IF xResetRequest//清空报警
THEN
	eERRORID := MT_MCK_ERROR.No_ERROR;
END_IF
IF  xAutoMode OR xDeviceRunning THEN
	xAutomodeFlag:=TRUE;
ELSE
	xAutomodeFlag:=FALSE;
END_IF


IF eErrorID = MT_MCK_ERROR.NO_ERROR AND xEStop 
THEN
//获取序列号
	IF(stDeviceOpe.xReadSerialNum_HMI AND NOT xAutomodeFlag) OR (stDeviceOpe.xReadSerialNum_Auto AND xAutomodeFlag) THEN
		eCmd := MT_MCK_CMD.Cmd_SerialNum;
		xExecute := TRUE;
	END_IF
//获取重量
	IF (stDeviceOpe.xAcquireWeight_Steady_HMI AND NOT xAutomodeFlag) OR (stDeviceOpe.xAcquireWeight_Steady_Auto AND xAutomodeFlag) THEN
		eCmd := MT_MCK_CMD.Cmd_AcquireWeight_Steady;
		xExecute := TRUE;		
	END_IF
	IF (stDeviceOpe.xAcquireWeight_RealTime_HMI AND NOT xAutomodeFlag) OR (stDeviceOpe.xAcquireWeight_RealTime_Auto AND xAutomodeFlag) THEN
		eCmd := MT_MCK_CMD.Cmd_AcquireWeight_RealTime;
		xExecute := TRUE;		
	END_IF	
	IF (stDeviceOpe.xAcquireWeight_Continuous_HMI AND NOT xAutomodeFlag) OR (stDeviceOpe.xAcquireWeight_Continuous_Auto AND xAutomodeFlag) THEN
		eCmd := MT_MCK_CMD.Cmd_AcquireWeight_Continuous;
		xExecute := TRUE;		
	END_IF	
	IF (stDeviceOpe.xAcquireWeight_Stop_HMI AND NOT xAutomodeFlag) OR (stDeviceOpe.xAcquireWeight_Stop_Auto AND xAutomodeFlag) THEN
		eCmd := MT_MCK_CMD.Cmd_AcquireWeight_Stop;
		xExecute := TRUE;		
	END_IF
//重启
	IF (stDeviceOpe.xRestart_HMI AND NOT xAutomodeFlag) OR (stDeviceOpe.xRestart_Auto AND xAutomodeFlag) THEN
		eCmd := MT_MCK_CMD.Cmd_Restart;
		xExecute := TRUE;		
	END_IF	
//去皮重
	IF (stDeviceOpe.xShelling_HMI AND NOT xAutomodeFlag) OR (stDeviceOpe.xShelling_Auto AND xAutomodeFlag) THEN
		eCmd := MT_MCK_CMD.Cmd_Shelling;
		xExecute := TRUE;		
	END_IF	
	IF (stDeviceOpe.xShellingInstanly_HMI AND NOT xAutomodeFlag) OR (stDeviceOpe.xShellingInstanly_Auto AND xAutomodeFlag) THEN
		eCmd := MT_MCK_CMD.Cmd_ShellingInstanly;
		xExecute := TRUE;		
	END_IF
	IF (stDeviceOpe.xSetTare_HMI AND NOT xAutomodeFlag) OR (stDeviceOpe.xSetTare_Auto AND xAutomodeFlag) THEN
		rTareSet:=stpar.rTarePresetValue;//
		eCmd := MT_MCK_CMD.Cmd_SetTare;
		xExecute := TRUE;		
	END_IF
	IF (stDeviceOpe.xlearTare_HMI AND NOT xAutomodeFlag) OR (stDeviceOpe.xlearTare_Auto AND xAutomodeFlag) THEN
		eCmd := MT_MCK_CMD.Cmd_ClearTare;
		xExecute := TRUE;		
	END_IF	
//清零
	IF (stDeviceOpe.xClearZero_HMI AND NOT xAutomodeFlag) OR (stDeviceOpe.xClearZero_Auto AND xAutomodeFlag) THEN
		eCmd := MT_MCK_CMD.Cmd_ClearZero;
		xExecute := TRUE;		
	END_IF	
	IF (stDeviceOpe.xClearZeroInstanly_HMI AND NOT xAutomodeFlag) OR (stDeviceOpe.xClearZeroInstanly_Auto AND xAutomodeFlag) THEN
		eCmd := MT_MCK_CMD.Cmd_ClearZeroInstanly;
		xExecute := TRUE;		
	END_IF		
	
END_IF
END_METHOD

{attribute 'tc_no_symbol'}
METHOD PRIVATE FINAL  HandleErrorSTATE
VAR_INPUT
END_VAR
VAR_OUTPUT
	xAgain: BOOL;
END_VAR
IF xError AND  (xResetRequest OR NOT xExecute) THEN
    eState:=STATE.RESETING;
    xAgain:=1;
ELSE
    xBusy:=0;
    xError:=1;    
    xAgain:=0;(* !!! *)
END_IF
END_METHOD

{attribute 'tc_no_symbol'}
METHOD PRIVATE FINAL HandleExecutingSTATE
VAR_INPUT
END_VAR
VAR_OUTPUT
	xAgain: BOOL;
END_VAR
VAR
{attribute 'tc_no_symbol'}	
	xComplete: BOOL;
END_VAR

IF xAbort=0 THEN   
    CyclicAction(xComplete=> xComplete);
END_IF

IF eErrorID<>MT_MCK_ERROR.NO_ERROR THEN
    eState:=STATE.INERROR;
    xAgain:=1;
ELSIF xAbort THEN
    eState:=STATE.ABORTING;
    xAgain:=1;
ELSIF xComplete THEN
    eState:=STATE.DONE;
    xAgain:=1;
END_IF
END_METHOD

{attribute 'tc_no_symbol'}
METHOD PRIVATE FINAL HandleResettingSTATE
VAR_INPUT
END_VAR
VAR_OUTPUT
	xAgain: BOOL;
END_VAR
VAR
{attribute 'tc_no_symbol'}	
	xComplete: BOOL;
END_VAR
ResetAction(xComplete=> xComplete);

IF xComplete THEN
		xExecute:=0;//清除输入指令 
    xBusy:=0;
    _xDone:=0;
    xError:=0;

    eErrorID:=MT_MCK_ERROR.NO_ERROR;
    eState:=STATE.DORMANT;
    xFirstInvocation:=1;
    xAgain:=0;(* !!! *)
END_IF
END_METHOD

{attribute 'tc_no_symbol'}
METHOD PROTECTED ResetAction
VAR_INPUT
END_VAR
VAR_OUTPUT
	xComplete: BOOL;
END_VAR
(*
* Cleaning
* => free all allocated resources
* => reinitialize instance variables
*)
tOperationTimer(IN:=0);
_tDelay(IN:=FALSE);
_iNGCount  := 0;
_fbTcpIpClient(xEnable:=FALSE);
_diCmdState:=0;
eCmd := MT_MCK_CMD.Nodef;

//复位操作按钮
	stDeviceOpe.xAcquireWeight_Continuous_Auto	:=
	stDeviceOpe.xAcquireWeight_Continuous_HMI	:=
	stDeviceOpe.xAcquireWeight_RealTime_Auto	:=
	stDeviceOpe.xAcquireWeight_RealTime_HMI		:=
	stDeviceOpe.xAcquireWeight_Steady_Auto		:=
	stDeviceOpe.xAcquireWeight_Steady_HMI		:=
	stDeviceOpe.xAcquireWeight_Stop_Auto		:=
	stDeviceOpe.xAcquireWeight_Stop_HMI			:=
	stDeviceOpe.xClearZero_Auto					:=
	stDeviceOpe.xClearZero_HMI                  :=
	stDeviceOpe.xClearZeroInstanly_Auto         :=
	stDeviceOpe.xClearZeroInstanly_HMI          :=
	stDeviceOpe.xlearTare_Auto                  :=
	stDeviceOpe.xlearTare_HMI                   :=
	stDeviceOpe.xReadSerialNum_Auto             :=
	stDeviceOpe.xReadSerialNum_HMI              :=
	stDeviceOpe.xRestart_Auto					:=
	stDeviceOpe.xRestart_HMI                    :=
	stDeviceOpe.xSetTare_Auto                   :=
	stDeviceOpe.xSetTare_HMI                    :=
	stDeviceOpe.xShelling_Auto                  :=
	stDeviceOpe.xShelling_HMI                   :=
	stDeviceOpe.xShellingInstanly_Auto          :=
	stDeviceOpe.xShellingInstanly_HMI           :=FALSE;

xComplete:=1;
END_METHOD

END_FUNCTION_BLOCK

// ---- POUs/003_FB/53_RudongPump/08_PeristalticPumpFB/校准程序/FB_AutoCal.TcPOU
{attribute 'tc_no_symbol'}
FUNCTION_BLOCK FB_AutoCal//METTLER电子秤
VAR_INPUT
	xExecute		: BOOL;//指令执行
	xAbort			: BOOL;//指令中断
	xEstop			: BOOL;//急停
	xDeviceRunning	: BOOL;
	xResetRequest	: BOOL;//复位操作
	stDeviceOpe		: ST_AutoCalOpe;
	stparIn				: STAutoCal_ParIn;	 
	stSysPar			: ST_AutoCal_SysPar; 
	xAutoMode    	: BOOL;//0:mannal 1:auto
	xIniting    	: BOOL;//初始化过程中  

END_VAR
VAR_OUTPUT
	xDone			: BOOL;(*完成条件满足*)
	xBusy			: BOOL;(*动作正在执行*)
	xRunning	: BOOL;
	xError			: BOOL;(*错误条件满足*)
	eERRORID		: AutoCal_ERROR;
	xRdyCmd			: BOOL;//指令就绪
	xRdy			: BOOL;//初始化完成
	sHmiError	:STRING;
	stParOut		: STAutoCal_ParOut;
END_VAR

VAR
{attribute 'tc_no_symbol'}
	eState: STATE;//当前状态
{attribute 'tc_no_symbol'}
	xAborted: BOOL;(*指令被打断，一般是处于急停中*)
{attribute 'tc_no_symbol'}
	_CalStep	:INT;//校准流程
{attribute 'tc_no_symbol'}
	_CurrentPumpController	:INT:=1;//当前控制器
{attribute 'tc_no_symbol'}
	_CurrentPumpHead	:INT:=1;//当前泵头
{attribute 'tc_no_symbol'}
	_first :BOOL;
{attribute 'tc_no_symbol'}		
	_xModeChange:BOOL;
{attribute 'tc_no_symbol'}
	_fManual:F_TRIG;
{attribute 'tc_no_symbol'}
	_rManual:R_TRIG;
{attribute 'tc_no_symbol'}	
	i:INT;
{attribute 'tc_no_symbol'}		
	xFirstInvocation:BOOL;
{attribute 'tc_no_symbol'}	
	xAutomodeFlag:BOOL;	
{attribute 'tc_no_symbol'}		
	_diCmdState:INT;
{attribute 'tc_no_symbol'}
	eCmd:AutoCal_CMD;
{attribute 'tc_no_symbol'}
	tOperationTimer:TON;
{attribute 'tc_no_symbol'}
	tSteadyTimer:TON;	
{attribute 'tc_no_symbol'}	
	_xAutoOpe:BOOL;
{attribute 'tc_no_symbol'}	
	_xHMIOpe:BOOL;
{attribute 'tc_no_symbol'}	
	_xDone:BOOL;
{attribute 'tc_no_symbol'}	
	_InjectNum	:INT;//
{attribute 'tc_no_symbol'}
	k	:INT;//
{attribute 'tc_no_symbol'}
	xRuDongPumpError	:BOOL;	
{attribute 'tc_no_symbol'}
OperR_TRIG:ARRAY[1..5] OF R_TRIG;	
END_VAR

VAR_TEMP
{attribute 'tc_no_symbol'}
	xAgain: BOOL;

END_VAR

VAR

END_VAR


IF NOT _first 
THEN
	_first := TRUE;

ELSE
	xAgain:=0;	
//检测是否允许指令控制(初始状态，没有报警发生)	
	xRdyCmd := eState = STATE.DORMANT AND eERRORID = AutoCal_ERROR.No_ERROR;
	xDone:=_xDone AND xExecute;	
	//检测是否有模式变化
_fManual(CLK:=xAutoMode);
_rManual(CLK:=xAutoMode);
//

IF eState <> STATE.DORMANT//只有在运行的时候，才会检测是否有模式切换发生
THEN
	IF _fManual.Q OR _rManual.Q
	THEN
		_xModeChange := TRUE;
	END_IF
END_IF
	REPEAT
		CASE eState OF
			STATE.DORMANT:
				HandleDormantState(xAgain=> xAgain);
			STATE.EXECUTING:
				HandleExecutingState(xAgain=> xAgain);
			STATE.DONE:
				HandleDoneState(xAgain=> xAgain);
			STATE.INERROR:
				HandleErrorState(xAgain=> xAgain);
			STATE.ABORTING:
				HandleAbortingState(xAgain=> xAgain);
			STATE.ABORTED:
				HandleAbortedState(xAgain=> xAgain);
			STATE.RESETING:
				HandleResettingState(xAgain=> xAgain);
			END_CASE
	UNTIL (xAgain=0)
	END_REPEAT
END_IF


//报错内容输出
CASE eERRORID OF
	AutoCal_ERROR.FLT_AutoMode:
		sHmiError:='FLT_AutoMode';
	AutoCal_ERROR.FLT_CmdTimeOut:
		sHmiError:='FLT_CmdTimeOut';	
	AutoCal_ERROR.FLT_MT_MCK204C:
		sHmiError:='FLT_MT_MCK204C';	
	AutoCal_ERROR.FLT_PARA:
		sHmiError:='FLT_PARA';	
	AutoCal_ERROR.FLT_RudongPump:
		sHmiError:='FLT_RudongPump';	
	AutoCal_ERROR.No_ERROR:
		sHmiError:='No_ERROR';
END_CASE




_xAutoOpe:=stDeviceOpe.x96PumpHeadCal_Auto OR
					stDeviceOpe.xSpecificPumpHeadCal_Auto;
_xHMIOpe:=stDeviceOpe.x96PumpHeadCal_HMI OR
					stDeviceOpe.xContinuesInject_HMI OR
					stDeviceOpe.xInit_Hmi OR
					stDeviceOpe.xSpecificPumpHeadCal_HMI;

{attribute 'tc_no_symbol'}
METHOD PROTECTED AbortAction
VAR_INPUT
END_VAR
VAR_OUTPUT
	xComplete: BOOL;
	eErrorID: AutoCal_ERROR;
END_VAR
(*
* Cleaning
* => abort all running operation
* => if an NBS.ERROR codition is reached, set eErrorID to a Value rather then NBS.ERROR.NO_ERROR 
*)
xComplete:=1;
eErrorID:=AutoCal_ERROR.NO_ERROR;
END_METHOD

ACTION ACT_DensityConversion:
{attribute 'tc_no_symbol'}
//密度计算公式，ρ＝m/V 
IF stParIn.rDensity<>0 THEN
	stParOut.rVolume:=stParOut.rSteadyWeight/stParIn.rDensity;
ELSE
	stParOut.rVolume:=0;
END_IF
END_ACTION

METHOD PROTECTED Cmd_ContinuesInject : BOOL
VAR_INPUT
END_VAR
VAR_OUTPUT
	xComplete: BOOL;
END_VAR
// return the real actual fault number
IF eERRORID <> AutoCal_ERROR.No_ERROR
THEN
  RETURN;  
END_IF
stParOut.iCalStep:=_diCmdState;//流程步输出

CASE _diCmdState OF	
	
		
	0://判断是否到达校准位置
		_diCmdState:=_diCmdState+1;	
			
	1://判断是否结束
	IF _InjectNum<=stparIn.iContinuesInjectNum THEN
		_diCmdState:=_diCmdState+1;
	ELSE
		_diCmdState:=30;//结束加液
	END_IF				
	
	2://等待秤Ready
		IF stsyspar.fbMTMCK204C^.xRdyCmd AND stsyspar.fbRuDongPump[stparIn.iPumpController-1].xRdyCmd THEN
			_diCmdState:=_diCmdState+1;	
		END_IF
	
	3://秤体清零
		stsyspar.fbMTMCK204C^.stDeviceOpe.xShelling_Auto:=TRUE;
			_diCmdState:=_diCmdState+1;
	4://等待清零完成
		IF stsyspar.fbMTMCK204C^.xQDone THEN
			_diCmdState:=_diCmdState+1;
		END_IF

	5://等待稳定时间
		tSteadyTimer(IN:=stsyspar.fbMTMCK204C^.xRdyCmd,PT:=T#1S);
		IF tSteadyTimer.Q THEN
			tSteadyTimer(IN:=FALSE);
			_diCmdState:=_diCmdState+1;
		END_IF	
	
	6://蠕动泵加液
		stsyspar.fbRuDongPump[stparIn.iPumpController-1].stDeviceOpe.xPush_Auto[1]:=TRUE;
		IF stsyspar.fbRuDongPump[stparIn.iPumpController-1].xDone THEN
			stsyspar.fbRuDongPump[stparIn.iPumpController-1].xExecute:=FALSE;
			_diCmdState:=_diCmdState+1;
		END_IF

	7://等待稳定时间
		tSteadyTimer(IN:=stsyspar.fbRuDongPump[stparIn.iPumpController-1].xRdyCmd,PT:=TO_TIME((stparIn.tSteadyTime +stsyspar.fbRuDongPump[stparIn.iPumpController-1].stRunPara.rPushRuntime[1])*1000 ));
		IF tSteadyTimer.Q THEN
			tSteadyTimer(IN:=FALSE);
			_diCmdState:=_diCmdState+1;
		END_IF
	
	8://读取重量
		stsyspar.fbMTMCK204C^.stDeviceOpe.xAcquireWeight_Steady_Auto:=TRUE;
			_diCmdState:=_diCmdState+1;
	9://等待读取完成
					IF stsyspar.fbMTMCK204C^.xQDone THEN
								_diCmdState:=_diCmdState+1;
					END_IF
	10://等待稳定时间
		tSteadyTimer(IN:=stsyspar.fbMTMCK204C^.xRdyCmd,PT:=T#1S);
		IF tSteadyTimer.Q THEN
			tSteadyTimer(IN:=FALSE);
			_diCmdState:=_diCmdState+1;
		END_IF		
		
	11://传递重量值
		IF stsyspar.fbMTMCK204C^.stParOut.rCurrentWeight>0 THEN
			stParOut.rContinuesInjectWeight[_InjectNum]:=stsyspar.fbMTMCK204C^.stParOut.rCurrentWeight;
			IF stParOut.rContinuesInjectWeight[_InjectNum]=stsyspar.fbMTMCK204C^.stParOut.rCurrentWeight THEN
				_diCmdState:=_diCmdState+1;
			END_IF
		ELSE
			_diCmdState:=8;
		END_IF		
	
	12://累加
		_InjectNum:=_InjectNum+1;
		_diCmdState:=_diCmdState+1;
	
	13://复位状态
		tSteadyTimer(IN:=TRUE,PT:=T#1S);
		IF tSteadyTimer.Q THEN
			tSteadyTimer(IN:=FALSE);
			_diCmdState:=0;
		END_IF	
		
		
(**************************************************加液结束***************************************************)	
	30://校准完成
		xComplete:=TRUE;
		
	
	
	
	
END_CASE
END_METHOD

METHOD PROTECTED Cmd_Init : BOOL
VAR_INPUT
END_VAR
VAR_OUTPUT
	xComplete: BOOL;
END_VAR
// return the real actual fault number
IF eERRORID <> AutoCal_ERROR.No_ERROR
THEN
  RETURN;  
END_IF
stParOut.iCalStep:=_diCmdState;//流程步输出
CASE _diCmdState OF	
		
	0://
		_CurrentPumpController:=1;//从1#泵开始
		_diCmdState:=10;
(**************蠕动泵停止**************)			
	10://判断N#泵控制器参数
		_CurrentPumpController:=1;//从1#开始
		_diCmdState:=_diCmdState+1;
		
	11://判断是否结束
		IF	_CurrentPumpController>=gc_uiRudongPump THEN
			_diCmdState:=20;
		ELSE
		 stSysPar.fbRuDongPump[_CurrentPumpController-1].xExecute:=FALSE;
			IF stSysPar.fbRuDongPump[_CurrentPumpController-1].xRdyCmd THEN
				_diCmdState:=_diCmdState+1;
			END_IF
		END_IF
		
	12://停止N#泵控制器	
		stSysPar.fbRuDongPump[_CurrentPumpController-1].stDeviceOpe.xStop_Auto:=TRUE;
				_diCmdState:=_diCmdState+1;
	13://等待停止	
					IF stSysPar.fbRuDongPump[_CurrentPumpController-1].xDone THEN
					 stSysPar.fbRuDongPump[_CurrentPumpController-1].stDeviceOpe.xStop_Auto:=FALSE;
						stSysPar.fbRuDongPump[_CurrentPumpController-1].xExecute:=FALSE;
						_diCmdState:=_diCmdState+1;
					END_IF	
	14://累加1
		_CurrentPumpController:=_CurrentPumpController+1;
		_diCmdState:=_diCmdState+1;
		
	15://回去循环执行
		_diCmdState:=11;

(**************************************************秤清零***************************************************)	
	20://判断秤体状态
		IF stSysPar.fbMTMCK204C^.xRdyCmd THEN
			_diCmdState:=22;
		ELSE
			IF stSysPar.fbMTMCK204C^.stParOut.xContinuesRead THEN
				_diCmdState:=_diCmdState+1;
			END_IF
		END_IF
	
	21://停止连续读取
			stSysPar.fbMTMCK204C^.stDeviceOpe.xAcquireWeight_Stop_Auto:=TRUE;
			IF stSysPar.fbMTMCK204C^.xRdyCmd THEN
				_diCmdState:=_diCmdState+1;
			END_IF			

	22://秤清零
			stSysPar.fbMTMCK204C^.stDeviceOpe.xClearZeroInstanly_Auto:=TRUE;
			_diCmdState:=_diCmdState+1;
	23://称清零完成
			IF stSysPar.fbMTMCK204C^.xQDone THEN
				_diCmdState:=30;
			END_IF			
	

(*************************************************初始化结束***************************************************)
	30://校准完成
		xComplete:=TRUE;
		

	
END_CASE
END_METHOD

METHOD PROTECTED Cmd_SpecificPumpHeadCal : BOOL
VAR_INPUT
END_VAR
VAR_OUTPUT
	xComplete: BOOL;
END_VAR
// return the real actual fault number
IF eERRORID <> AutoCal_ERROR.No_ERROR
THEN
  RETURN;  
END_IF
stParOut.iCalStep:=_diCmdState;//流程步输出

CASE _diCmdState OF	
	
		
	0://判断是否到达校准位置
		_diCmdState:=_diCmdState+1;	
		
	1://等待校准就绪
		stsyspar.fbRuDongPump[stparIn.iPumpController-1].xExecute:=FALSE;
		IF stsyspar.fbMTMCK204C^.xQRdyCmd AND stsyspar.fbRuDongPump[stparIn.iPumpController-1].xRdyCmd THEN
			_diCmdState:=_diCmdState+1;	

		END_IF		
		
(**************************************************校准***************************************************)		
	2://秤体清零	
		stSysPar.fbMTMCK204C^.stDeviceOpe.xClearZero_Auto:=TRUE;
			_diCmdState:=_diCmdState+1;	
	3://清零完成
		IF stSysPar.fbMTMCK204C^.xQDone THEN
			_diCmdState:=_diCmdState+1;	
		END_IF
		
	4://等待稳定时间
		tSteadyTimer(IN:=TRUE,PT:=T#1S);
		IF tSteadyTimer.Q THEN
			tSteadyTimer(IN:=FALSE);
			_diCmdState:=_diCmdState+1;
		END_IF		
		
	5://校准启动
		stSysPar.fbRuDongPump[_CurrentPumpController-1].stDeviceOpe.xPumpCal_Auto:=TRUE;
		IF stSysPar.fbRuDongPump[_CurrentPumpController-1].xDone THEN
		 	stSysPar.fbRuDongPump[_CurrentPumpController-1].xExecute:=FALSE;
			_diCmdState:=_diCmdState+1;
		END_IF
		
	6://等待稳定时间
		tSteadyTimer(IN:=TRUE,PT:=TO_TIME((stparIn.tSteadyTime+1)*1000));
		IF tSteadyTimer.Q THEN
			_diCmdState:=_diCmdState+1;
		END_IF

	7://获取称重结果
			stSysPar.fbMTMCK204C^.stDeviceOpe.xAcquireWeight_Steady_Auto:=TRUE;
				_diCmdState:=_diCmdState+1;
	8://等待完成
			IF stSysPar.fbMTMCK204C^.xQDone THEN
				_diCmdState:=_diCmdState+1;	
			END_IF	
	
	9://等待稳定时间
		tSteadyTimer(IN:=TRUE,PT:=T#1S);
		IF tSteadyTimer.Q THEN
			tSteadyTimer(IN:=FALSE);
			_diCmdState:=_diCmdState+1;
		END_IF			

	10://获取称重结果
		IF stSysPar.fbMTMCK204C^.stParOut.rCurrentWeight>0 THEN
			stParOut.rSteadyWeight:=stSysPar.fbMTMCK204C^.stParOut.rCurrentWeight;
			IF stParOut.rSteadyWeight=stSysPar.fbMTMCK204C^.stParOut.rCurrentWeight THEN
				_diCmdState:=_diCmdState+1;
			END_IF
		ELSE
			_diCmdState:=7;//未获取到重量重新读
		END_IF
		
	11://给校准参数赋值
		stSysPar.fbRuDongPump^.stRunPara.rModuleRealFluVolume:=stParOut.rVolume;
		stSysPar.fbRuDongPump^.stDeviceOpe.xCalParWrite_Auto:=TRUE;
		IF stSysPar.fbRuDongPump^.xDone THEN
			_diCmdState:=30;
		END_IF
	

(**************************************************校准结束***************************************************)	
	30://校准完成
		xComplete:=TRUE;
		
	
	
	
	
END_CASE
END_METHOD

{attribute 'tc_no_symbol'}
METHOD PROTECTED CyclicAction
VAR_INPUT
END_VAR
VAR_OUTPUT
	xComplete: BOOL;
END_VAR
VAR	
END_VAR
IF xAbort=0 THEN
	IF xFirstInvocation THEN//执行初始化
	(*
	* Staring
	* for then first (!) invocaion,
	* sample then input variables
	*)
		xFirstInvocation:=0;
	END_IF    
	REPEAT 	
//判断是否有参数错误		
		IF stSysPar.fbMTMCK204C=0 OR
				stSysPar.fbRuDongPump=0 OR
				stSysPar.iRuDongPumpHeadNum>32
		THEN
			eERRORID:=AutoCal_ERROR.FLT_PARA;//参数配置错误
		ELSE
			xRuDongPumpError:=FALSE;
			FOR k:=1 TO gc_uiRudongPump DO
				IF stSysPar.fbRuDongPump[k].xError THEN
					xRuDongPumpError:=TRUE;
					EXIT;
				END_IF
			END_FOR			

			//IF stSysPar.fbMTMCK204C^.xError THEN
			//	eERRORID:=AutoCal_ERROR.FLT_MT_MCK204C;//秤出错
			//ELSE
			//	IF xRuDongPumpError THEN
			//		eERRORID:=AutoCal_ERROR.FLT_RudongPump;//蠕动泵出错
			//	END_IF						
			//END_IF
		END_IF

			//如果不在自动模式则报错
			IF _xAutoOpe OR _xHMIOpe THEN
					xRunning:=TRUE;
			END_IF

			CASE eCmd OF//判断指令类型
				AutoCal_CMD.Cmd_SpecificPumpHeadCal://单个泵头校准
					Cmd_SpecificPumpHeadCal(xComplete=> xComplete);	
				AutoCal_CMD.Cmd_Init://初始化
					Cmd_Init(xComplete=> xComplete);	
				AutoCal_CMD.Cmd_ContinuesInject://连续加液测试
					Cmd_ContinuesInject(xComplete=> xComplete);
					;				
				
			ELSE
				;	
			END_CASE
	   
		UNTIL (TRUE)//处于一直刷新阶段
	END_REPEAT
END_IF

IF NOT xExecute OR xComplete OR eErrorID<>AutoCal_ERROR.No_ERROR THEN    
    (*
    * Cleaning
    * => free as much allocated resources as possible
    *)    
    tOperationTimer(IN:=0);
END_IF
END_METHOD

{attribute 'tc_no_symbol'}
METHOD PRIVATE FINAL HandleAbortedSTATE
VAR_INPUT
END_VAR
VAR_OUTPUT
	xAgain: BOOL;
END_VAR
VAR
	xComplete: BOOL;
END_VAR
IF xAborted AND xResetRequest THEN
    eState:=STATE.RESETING;
    xAgain:=1;
ELSE
    xBusy:=0;
    xAborted:=1;
    //xResetRequest:=(xExecute=0);
    xAgain:=0;(* !!! *)
END_IF
END_METHOD

{attribute 'tc_no_symbol'}
METHOD PRIVATE FINAL HandleAbortingSTATE
VAR_INPUT
END_VAR
VAR_OUTPUT
	xAgain: BOOL;
END_VAR
VAR
{attribute 'tc_no_symbol'}	
	xComplete: BOOL;
END_VAR
AbortAction(xComplete=> xComplete, eErrorID=> eErrorID);

IF eErrorID<>AutoCal_ERROR.NO_ERROR THEN
    eState:=STATE.INERROR;
    xAgain:=1;
ELSIF xComplete THEN
    eState:=STATE.ABORTED;
    xAgain:=1;
END_IF
END_METHOD

{attribute 'tc_no_symbol'}
METHOD PRIVATE FINAL HandleDoneSTATE
VAR_INPUT
END_VAR
VAR_OUTPUT
	xAgain: BOOL;
END_VAR
//在运行过程中要是切换模式，再运行完成之后，检测到模式的切换，就需要回到初始位置，进行下一次执行准备
IF _xDone AND ((xExecute=0) OR ( _xModeChange AND NOT _xAutoOpe)  OR ( NOT xAutoMode AND NOT xDeviceRunning AND ( NOT _xAutoOpe OR _xHMIOpe))) THEN
	eState:=STATE.RESETING;
	xAgain:=1;
ELSE
	xBusy:=0;
	_xDone:=1;
	//xResetRequest:=(xExecute=0);
	xAgain:=0;(* !!! *)
END_IF
END_METHOD

{attribute 'tc_no_symbol'}
METHOD PRIVATE FINAL HandleDormantSTATE
VAR_INPUT
END_VAR
VAR_OUTPUT
	xAgain: BOOL;
END_VAR
IF xExecute THEN
    xBusy:=1;
    eState:=STATE.EXECUTING;
    xAgain:=1;
END_IF

IF xResetRequest//清空报警
THEN
	eERRORID := AutoCal_ERROR.No_ERROR;
END_IF
IF  xAutoMode OR xDeviceRunning THEN
	xAutomodeFlag:=TRUE;
ELSE
	xAutomodeFlag:=FALSE;
END_IF
(********************************等待手动操作******************************)
OperR_TRIG[1](CLK:=  (stDeviceOpe.xSpecificPumpHeadCal_HMI OR stDeviceOpe.xSpecificPumpHeadCal_Auto) , Q=> );
OperR_TRIG[2](CLK:=  (stDeviceOpe.xInit_Hmi  OR stDeviceOpe.xInit_Auto)  , Q=> );

IF eErrorID = AutoCal_ERROR.NO_ERROR AND xEStop
THEN
	
//校准指定泵头
	IF OperR_TRIG[1].Q THEN//
		_CurrentPumpController:=stparIn.iPumpController;
		_CurrentPumpHead:=stparIn.iPumpHead;
		eCmd := AutoCal_CMD.Cmd_SpecificPumpHeadCal;
		xExecute := TRUE;
	END_IF
//初始化校准程序
	IF OperR_TRIG[2].Q THEN//
		eCmd := AutoCal_CMD.Cmd_Init;
		xExecute := TRUE;
	END_IF	
	
	
	
	stDeviceOpe.xSpecificPumpHeadCal_HMI := stDeviceOpe.xSpecificPumpHeadCal_Auto:=FALSE;
	stDeviceOpe.xInit_Hmi  := stDeviceOpe.xInit_Auto:=FALSE;
	
//连续加液测试
	IF stDeviceOpe.xContinuesInject_HMI THEN//
		FOR i:=1 TO 30 DO
			stParOut.rContinuesInjectWeight[i]:=0;
		END_FOR
		_InjectNum:=1;
		eCmd := AutoCal_CMD.Cmd_ContinuesInject;
		xExecute := TRUE;
	END_IF	
	
END_IF
END_METHOD

{attribute 'tc_no_symbol'}
METHOD PRIVATE FINAL  HandleErrorSTATE
VAR_INPUT
END_VAR
VAR_OUTPUT
	xAgain: BOOL;
END_VAR
IF xError AND  (xResetRequest OR NOT xExecute) THEN
    eState:=STATE.RESETING;
    xAgain:=1;
ELSE
    xBusy:=0;
    xError:=1;    
    xAgain:=0;(* !!! *)
END_IF
END_METHOD

{attribute 'tc_no_symbol'}
METHOD PRIVATE FINAL HandleExecutingSTATE
VAR_INPUT
END_VAR
VAR_OUTPUT
	xAgain: BOOL;
END_VAR
VAR
{attribute 'tc_no_symbol'}	
	xComplete: BOOL;
END_VAR

IF xAbort=0 THEN   
    CyclicAction(xComplete=> xComplete);
END_IF

IF eErrorID<>AutoCal_ERROR.NO_ERROR THEN
    eState:=STATE.INERROR;
    xAgain:=1;
ELSIF xAbort THEN
    eState:=STATE.ABORTING;
    xAgain:=1;
ELSIF xComplete THEN
    eState:=STATE.DONE;
    xAgain:=1;
END_IF
END_METHOD

{attribute 'tc_no_symbol'}
METHOD PRIVATE FINAL HandleResettingSTATE
VAR_INPUT
END_VAR
VAR_OUTPUT
	xAgain: BOOL;
END_VAR
VAR
{attribute 'tc_no_symbol'}	
	xComplete: BOOL;
END_VAR
ResetAction(xComplete=> xComplete);

IF xComplete THEN
		xExecute:=0;//清除输入指令 
    xBusy:=0;
    xDone:=0;
    xError:=0;

    eErrorID:=AutoCal_ERROR.NO_ERROR;
    eState:=STATE.DORMANT;
    xFirstInvocation:=1;
    xAgain:=0;(* !!! *)
END_IF
END_METHOD

{attribute 'tc_no_symbol'}
METHOD PROTECTED ResetAction
VAR_INPUT
END_VAR
VAR_OUTPUT
	xComplete: BOOL;
END_VAR
(*
* Cleaning
* => free all allocated resources
* => reinitialize instance variables
*)
tOperationTimer(IN:=0);
_diCmdState:=0;
_CurrentPumpController:=1;
stDeviceOpe.x96PumpHeadCal_Auto:=
stDeviceOpe.x96PumpHeadCal_HMI:=
stDeviceOpe.xInit_Auto:=
stDeviceOpe.xInit_Hmi:=
stDeviceOpe.xSpecificPumpHeadCal_Auto:=
stDeviceOpe.xContinuesInject_HMI:=
stDeviceOpe.xSpecificPumpHeadCal_HMI:=FALSE;
xRunning:=FALSE; 
xComplete:=1;	

stsyspar.fbRuDongPump[stparIn.iPumpController-1].xExecute:=FALSE;
//stsyspar.fbRuDongPump[stparIn.iPumpController-1].stDeviceOpe.xPush_Auto[1]:=TRUE;
stsyspar.fbRuDongPump[stparIn.iPumpController-1].stDeviceOpe.xStop_Auto:=TRUE;
END_METHOD

END_FUNCTION_BLOCK

// ---- POUs/003_FB/0015_Functions/FC_BubbleSort_Max.TcPOU
FUNCTION FC_BubbleSort_Max : REAL
(*
********************************************************************************
* Name: FB_BubbleSort_Max
*
* Author:  Automanh
* Version: 1.0.0
*
* Description:
*     将数组元素从小到大排列
*
* Remarks:
*
* Revisions:
*   1.0 -AutomanH Rebuild
*         
*  
*********************************************************************************)
VAR_INPUT
 i_i_Counter:INT;
 i_arrReal:ARRAY[1..3] OF REAL;
END_VAR
VAR
 i,j:INT;
 rRealTemp:REAL;
END_VAR


FOR i:=1 TO (i_i_Counter-1) BY 1 DO//控制比较轮次，一共 n-1 趟
 		FOR  j:=1 TO i_i_Counter-i BY 1 DO//控制两个挨着的元素进行比较
		 			IF i_arrReal[j]>i_arrReal[j+1] THEN
					 			rRealTemp:=i_arrReal[j];
								i_arrReal[j]:=i_arrReal[j+1];
								i_arrReal[j+1]:=rRealTemp;
					END_IF
		END_FOR
					
END_FOR
FC_BubbleSort_Max:=i_arrReal[i_i_Counter];

END_FUNCTION

// ---- POUs/003_FB/0015_Functions/FC_BubbleSort_Min.TcPOU
FUNCTION FC_BubbleSort_Min : REAL
(*
********************************************************************************
* Name: FB_BubbleSort_Min
*
* Author:  Automanh
* Version: 1.0.0
*
* Description:
*     将数组元素从大到小排列
*
* Remarks:
*
* Revisions:
*   1.0 -AutomanH Rebuild
*         
*  
*********************************************************************************)
VAR_INPUT
 i_i_Counter:INT;
 i_arrReal:ARRAY[1..3] OF REAL;
END_VAR
VAR
 i,j:INT;
 rRealTemp:REAL;
END_VAR

FOR i:=1 TO (i_i_Counter-1) BY 1 DO//控制比较轮次，一共 n-1 趟
 		FOR  j:=1 TO i_i_Counter-i BY 1 DO//控制两个挨着的元素进行比较
		 			IF i_arrReal[j]<i_arrReal[j+1] THEN
					 			rRealTemp:=i_arrReal[j];
								i_arrReal[j]:=i_arrReal[j+1];
								i_arrReal[j+1]:=rRealTemp;
					END_IF
		END_FOR
					
END_FOR
FC_BubbleSort_Min:=i_arrReal[i_i_Counter];

END_FUNCTION

// ---- POUs/001_Station/S03_LidChecking.TcPOU
PROGRAM S03_LidChecking
VAR
	//工站
	station					: REFERENCE TO FB_Station:=fbstation[3];
	//气缸
	fbHOZAdjustCyl_1	:REFERENCE TO FB_Cylinder:=fbCylinder[12];	//	上层水平调整气缸1（小）
	fbHOZAdjustCyl_2	:REFERENCE TO FB_Cylinder:=fbCylinder[13];	//	上层水平调整气缸2（小）
	fbHOZAdjustCyl_3	:REFERENCE TO FB_Cylinder:=fbCylinder[14];	//	下层水平调整气缸1（小）
	fbHOZAdjustCyl_4	:REFERENCE TO FB_Cylinder:=fbCylinder[15];	//	下层水平调整气缸2（小）
	fbHOZAdjustCyl_5	:REFERENCE TO FB_Cylinder:=fbCylinder[16];	//	上层水平调整气缸1（大）
	fbHOZAdjustCyl_6	:REFERENCE TO FB_Cylinder:=fbCylinder[17];	//	上层水平调整气缸2（大）
	fbHOZAdjustCyl_7	:REFERENCE TO FB_Cylinder:=fbCylinder[18];	//	下层水平调整气缸1（大）
	fbHOZAdjustCyl_8	:REFERENCE TO FB_Cylinder:=fbCylinder[19];	//	下层水平调整气缸2（大）
	//伺服
	fbXAxisMove	 :REFERENCE TO FB_Axis:=fbAxis[6];	//	相机检测工位X轴伺服
	fbYAxisMove	 :REFERENCE TO FB_Axis:=fbAxis[7];	//	相机检测工位Y轴伺服
	fbZAxisMove	 :REFERENCE TO FB_Axis:=fbAxis[8];	//	相机检测工位Z轴伺服
	//相机

	
		//延时
		arTonDelay :ARRAY[1..20] OF TON;
	//返回值
		UdiReturnValue :ARRAY[1..20] OF UDINT;
	//本地过程数据
	arProcessDataStation : ARRAY [1..5] OF DUT_MainlineFixture;
	
	i,j,k: INT;
	//循环使用
	i_b_REPEAT:BOOL;
	i_i_Counter:INT;
	//相机拍照结果步骤
	bResultStep:BYTE;
	// 循环计数
	bCounter: BYTE;
	// 临时变量
	_FirstCycle:ARRAY[1..10] OF BOOL;
	them: INT;
	// X轴伺服循环次数
	bXCounter: BYTE;
	// Y轴伺服循环次数
	bYCounter: BYTE;
	// 结束时循环次数
	bEndCounter: INT;
	//相机检测工位检测结果
	arCameraResult:ARRAY[1..5,1..4,1..12] OF INT;
	//过程记录
	tsModuleProcess:ARRAY[1..gc_ModuleProNo] OF DUT_Process;
	xClearModuleProcessDone:BOOL;
	bClearProcessStep	:BYTE;
	// 测试使用，待删
	xtest: BOOL;
	// //待删
	xnext: BOOL;
END_VAR

A_Input();
Alarm();
Delay();
FlowAuto();
FlowInit();
General();
ILC();
TipAuto();
TipManual();
Z_Output();

ACTION A_Input:
//气缸
//S03上层水平调整气缸1(小)
fbHOZAdjustCyl_1.xWP_Sensor	:=	IxS03HOZAdjustCyl_1WP	;
fbHOZAdjustCyl_1.xHP_Sensor	:=	IxS03HOZAdjustCyl_1HP 	;
//	上层水平调整气缸2（小）
fbHOZAdjustCyl_2.xWP_Sensor	:=	IxS03HOZAdjustCyl_2WP ;
fbHOZAdjustCyl_2.xHP_Sensor	:=	IxS03HOZAdjustCyl_2HP 	;

//S03下层水平调整气缸1(小)
fbHOZAdjustCyl_3.xWP_Sensor	:=	IxS03HOZAdjustCyl_5WP	;  
fbHOZAdjustCyl_3.xHP_Sensor	:=	IxS03HOZAdjustCyl_5HP ;
//下层水平调整气缸2（小）
fbHOZAdjustCyl_4.xWP_Sensor	:=	  IxS03HOZAdjustCyl_6WP;  
fbHOZAdjustCyl_4.xHP_Sensor	:=	  IxS03HOZAdjustCyl_6HP;
  
//S03上层水平调整气缸1(大）
fbHOZAdjustCyl_5.xWP_Sensor	:=IxS03HOZAdjustCyl_3WP ;										
fbHOZAdjustCyl_5.xHP_Sensor	:=IxS03HOZAdjustCyl_3HP	; 
//	上层水平调整气缸2（大）
fbHOZAdjustCyl_6.xWP_Sensor	:=IxS03HOZAdjustCyl_4WP ;										
fbHOZAdjustCyl_6.xHP_Sensor	:=IxS03HOZAdjustCyl_4HP	; 

//S03下层水平调整气缸1(大） 									 
fbHOZAdjustCyl_7.xWP_Sensor	:=	IxS03HOZAdjustCyl_7WP	;  
fbHOZAdjustCyl_7.xHP_Sensor	:=	IxS03HOZAdjustCyl_7HP	;  
//	下层水平调整气缸2（大）
fbHOZAdjustCyl_8.xWP_Sensor	:=		IxS03HOZAdjustCyl_8WP;  
fbHOZAdjustCyl_8.xHP_Sensor	:=		IxS03HOZAdjustCyl_8HP;
END_ACTION

ACTION Alarm:
station.adwAlarm[1].00	:=	station.xInitTimeout	;//	S03 初始化超时
station.adwAlarm[1].01	:=	fbHOZAdjustCyl_1.xHP_Off 	;//	S03上层水平调整气缸1(小)原点未到位
station.adwAlarm[1].02	:=	fbHOZAdjustCyl_1.xWP_Off 	;//	S03上层水平调整气缸1(小)动点未到位
station.adwAlarm[1].03	:=	fbHOZAdjustCyl_3.xHP_Off	;//	S03下层水平调整气缸1(小)原点未到位
station.adwAlarm[1].04	:=	fbHOZAdjustCyl_3.xWP_Off	;//	S03下层水平调整气缸1(小)动点未到位
station.adwAlarm[1].05	:=	fbHOZAdjustCyl_5.xHP_Off	;//	S03上层水平调整气缸1(大)原点未到位
station.adwAlarm[1].06	:=	fbHOZAdjustCyl_5.xWP_Off	;//	S03上层水平调整气缸1(大)动点未到位
station.adwAlarm[1].07	:=	fbHOZAdjustCyl_7.xHP_Off	;//	S03下层水平调整气缸1(大)原点未到位
station.adwAlarm[1].08	:=	fbHOZAdjustCyl_7.xWP_Off	;//	S03下层水平调整气缸1(大)动点未到位
station.adwAlarm[1].09	:=	fbXAxisMove.xError	;//	S03液位检测X轴伺服报错
station.adwAlarm[1].10	:=	fbXAxisMove.xNotPowerOn	;//	S03液位检测X轴伺服未使能
station.adwAlarm[1].11	:=	fbXAxisMove.xMoveTimeout	;//	S03液位检测X轴伺服移动超时
station.adwAlarm[1].12	:=	fbYAxisMove.xError	;//	S03液位检测Y轴伺服报错
station.adwAlarm[1].13	:=	fbYAxisMove.xNotPowerOn	;//	S03液位检测Y轴伺服未使能
station.adwAlarm[1].14	:=	fbYAxisMove.xMoveTimeout	;//	S03液位检测Y轴伺服移动超时
station.adwAlarm[1].15	:=	fbZAxisMove.xError	;//	S03液位检测Z轴伺服报错
station.adwAlarm[1].16	:=	fbZAxisMove.xNotPowerOn	;//	S03液位检测Z轴伺服未使能
station.adwAlarm[1].17	:=	fbZAxisMove.xMoveTimeout	;//	S03液位检测Z轴伺服移动超时
//station.adwAlarm[1].18	:=	true;//	S03液位检测工位-相机检测超时报警,请检查
END_ACTION

ACTION Delay:
arTonDelay[01](IN:= , PT:=T#0.1S , Q=> , ET=> );
arTonDelay[02](IN:=  , PT:=T#1S , Q=> , ET=> );
arTonDelay[03](IN:=   , PT:=T#1S , Q=> , ET=> );
arTonDelay[04](IN:= , PT:=T#0.1S , Q=> , ET=> );
arTonDelay[05](IN:= , PT:=T#0.1S , Q=> , ET=> );
arTonDelay[06](IN:= , PT:=T#0.1S , Q=> , ET=> );
(*arTonDelay[07](IN:= , PT:=T#200MS , Q=> , ET=> );*)//已使用
arTonDelay[08](IN:=NOT fbXAxisMove.xbusy , PT:=T#0.1S , Q=> , ET=> );//TipAuto使用
arTonDelay[09](IN:= NOT fbYAxisMove.xbusy, PT:=T#0.1S , Q=> , ET=> );//TipAuto使用
arTonDelay[10](IN:=NOT fbZAxisMove.xbusy , PT:=T#0.1S , Q=> , ET=> );//TipAuto使用
END_ACTION

ACTION FlowAuto:

//-----------------------------------------初始化是否完成判断----------------------------------------------
IF NOT station.xInitDone 
THEN
 	station.iStepAuto:=0;
 	station.xDone:=FALSE;
	station.xRunningOffProhibit := FALSE ;//运行中信号Off禁止
ELSIF station.xRunning // OR (tsModuleProcess[bXCounter+1].xProcessStarted AND NOT tsModuleProcess[bXCounter+1].xProcessCompleted )//相机检测流程
THEN
//-----------------------------------------动作步骤--------------------------------------------------------
CASE station.iStepAuto OF	  
	0: //----Home Step，等待启动----
		IF station.xDisabled 
			AND station.xCanRun 
			AND NOT fbMachine[1].xStopped 
			AND NOT station.xSingleRunning 
		THEN
			station.xDone:=TRUE;
		END_IF
		
		IF  station.xSingleRunning 
			OR station.xCanRun 
			AND NOT station.xDone 
			AND NOT station.xDisabled 
			AND NOT fbMachine[1].xStopped
		THEN
			station.xCycleEnable:=TRUE;
			station.xDone:= FALSE;  
			station.iStepAuto:= 5;
		END_IF		
	 5://复位数据
			FOR i:=1 TO gc_ModuleProNo BY 1 DO
				 MEMSET(ADR(tsModuleProcess[i]),0,SIZEOF(tsModuleProcess[i]));
			END_FOR
			station.iStepAuto:= 10;
	 10: //判断产品是否到该工位
		IF  station.xSingleRunning THEN
			station.iStepAuto:= 11;
		ELSE
		 			IF    station.xEmptyDone THEN
										station.iStepAuto:= 999;		
					//清料程序
					ELSIF   arMainlineFixtureData[arCurFixtureNumStation[5]].stProduct.xEmptying AND    
				    	arMainlineFixtureData[arCurFixtureNumStation[6]].stProduct.xEmptying  AND 
							arMainlineFixtureData[arCurFixtureNumStation[7]].xMaterialOnOff AND 
							arMainlineFixtureData[arCurFixtureNumStation[8]].xMaterialOnOff AND
							arMainlineFixtureData[arCurFixtureNumStation[9]].xMaterialOnOff  THEN
										 bEndCounter:=1;
										 bCounter:=0;
								 		 station.iStepAuto:= 11;
					ELSIF   arMainlineFixtureData[arCurFixtureNumStation[5]].stProduct.xEmptying AND    
									arMainlineFixtureData[arCurFixtureNumStation[6]].stProduct.xEmptying  AND 
									arMainlineFixtureData[arCurFixtureNumStation[7]].stProduct.xEmptying AND 
									arMainlineFixtureData[arCurFixtureNumStation[8]].stProduct.xEmptying AND
									arMainlineFixtureData[arCurFixtureNumStation[9]].xMaterialOnOff  THEN
												 bEndCounter:=2;
												 bCounter:=0;
												 station.iStepAuto:= 11;							 
					ELSIF   arMainlineFixtureData[arCurFixtureNumStation[5]].stProduct.xEmptying AND    
									arMainlineFixtureData[arCurFixtureNumStation[6]].stProduct.xEmptying  AND 
									arMainlineFixtureData[arCurFixtureNumStation[7]].stProduct.xEmptying AND 
									arMainlineFixtureData[arCurFixtureNumStation[8]].stProduct.xEmptying AND
									arMainlineFixtureData[arCurFixtureNumStation[9]].stProduct.xEmptying  THEN
												 station.xEmptying:=TRUE;
												 station.iStepAuto:= 1010;														
			//正常程序
				 ELSIF   NOT  arMainlineFixtureData[arCurFixtureNumStation[5]].xMaterialOnOff AND
								 NOT arMainlineFixtureData[arCurFixtureNumStation[6]].xMaterialOnOff  AND 
								 NOT arMainlineFixtureData[arCurFixtureNumStation[7]].xMaterialOnOff AND 
								 NOT	arMainlineFixtureData[arCurFixtureNumStation[8]].xMaterialOnOff AND
								 NOT arMainlineFixtureData[arCurFixtureNumStation[9]].xMaterialOnOff  THEN
											bCounter:=0;
											bEndCounter :=0;
											_FirstCycle[6]:=FALSE;
											station.iStepAuto:= 999;
				 ELSIF	 arMainlineFixtureData[arCurFixtureNumStation[5]].xMaterialOnOff AND    
							 arMainlineFixtureData[arCurFixtureNumStation[6]].xMaterialOnOff  AND 
							 NOT arMainlineFixtureData[arCurFixtureNumStation[7]].xMaterialOnOff AND 
							 NOT	arMainlineFixtureData[arCurFixtureNumStation[8]].xMaterialOnOff AND
							 NOT arMainlineFixtureData[arCurFixtureNumStation[9]].xMaterialOnOff   THEN
												bCounter:=1;
												bEndCounter :=0;
												station.iStepAuto:= 11;
				ELSIF	arMainlineFixtureData[arCurFixtureNumStation[5]].xMaterialOnOff AND    
							 arMainlineFixtureData[arCurFixtureNumStation[6]].xMaterialOnOff  AND 
							 arMainlineFixtureData[arCurFixtureNumStation[7]].xMaterialOnOff AND 
							 arMainlineFixtureData[arCurFixtureNumStation[8]].xMaterialOnOff AND
							 NOT arMainlineFixtureData[arCurFixtureNumStation[9]].xMaterialOnOff   THEN
												 bCounter:=2;
												 bEndCounter :=0;
												 station.iStepAuto:= 11;
				ELSIF  arMainlineFixtureData[arCurFixtureNumStation[5]].xMaterialOnOff AND      
							 arMainlineFixtureData[arCurFixtureNumStation[6]].xMaterialOnOff  AND 
							 arMainlineFixtureData[arCurFixtureNumStation[7]].xMaterialOnOff AND 
							 arMainlineFixtureData[arCurFixtureNumStation[8]].xMaterialOnOff AND
							 arMainlineFixtureData[arCurFixtureNumStation[9]].xMaterialOnOff   THEN
												 bCounter:=3;
												 bEndCounter :=0;
												 station.iStepAuto:= 11;
			 END_IF
	END_IF
	11://手动NOK按钮
			IF   arManualNOKHmiButton[3]  AND NOT station.xSingleRunning THEN
				station.iStepAuto:= 280;
			ELSE	
				station.iStepAuto:= 20;
			END_IF

	20:////Restore_after_Estop_Process1 上载数据流程
			IF   station.xSingleRunning  THEN//OR  fbMachine[1].xTryRun THEN
				    station.iStepAuto :=40;
			ELSIF tsModuleProcess[1].xProcessNotStarted AND NOT  tsModuleProcess[1].xProcessStarted THEN
					station.iStepAuto :=21; (*process not started*)
			ELSIF  tsModuleProcess[1].xProcessStarted AND NOT  tsModuleProcess[1].xProcessCompleted THEN
				 station.iStepAuto := 21;(*process started*)
			ELSIF  tsModuleProcess[1].xProcessCompleted AND NOT tsModuleProcess[1].xQDataCompleted  THEN
					station.iStepAuto := 40 ;(*process completed*)
			ELSIF tsModuleProcess[1].xQDataCompleted THEN
					station.iStepAuto :=40;(*Qdata completed *)
			ELSE
					station.iStepAuto :=21; 
			END_IF	
	21://
				tsModuleProcess[1].xProcessNotStarted:=TRUE;
				station.iStepAuto:= 30;
	30://上载产品数据
			tsModuleProcess[1].xProcessStarted	:=TRUE;
			IF  bCounter =1 OR bCounter =2 OR bCounter=3 THEN
				MEMCPY(ADR(arProcessDataStation[1]),ADR(arMainlineFixtureData[arCurFixtureNumStation[5]]),SIZEOF(arMainlineFixtureData[arCurFixtureNumStation[5]]));
				MEMCPY(ADR(arProcessDataStation[2]),ADR(arMainlineFixtureData[arCurFixtureNumStation[6]]),SIZEOF(arMainlineFixtureData[arCurFixtureNumStation[6]]))	;
			END_IF
			IF bCounter =2 OR bCounter =3 OR bEndCounter =1 THEN
				MEMCPY(ADR(arProcessDataStation[3]),ADR(arMainlineFixtureData[arCurFixtureNumStation[7]]),SIZEOF(arMainlineFixtureData[arCurFixtureNumStation[7]]));
				MEMCPY(ADR(arProcessDataStation[4]),ADR(arMainlineFixtureData[arCurFixtureNumStation[8]]),SIZEOF(arMainlineFixtureData[arCurFixtureNumStation[8]]))	;
			END_IF
			IF bCounter =3 OR bEndCounter =2 THEN
				MEMCPY(ADR(arProcessDataStation[5]),ADR(arMainlineFixtureData[arCurFixtureNumStation[9]]),SIZEOF(arMainlineFixtureData[arCurFixtureNumStation[9]]))	;
			END_IF
			tsModuleProcess[1].xProcessCompleted:=TRUE;
			station.iStepAuto:= 40;
	/////产品流程开始	
		40://设定X轴循环为1，总次数2
				 bXCounter:=1;
				station.iStepAuto:= 45;		
		45://测试所用
					//以下为测试所用
					IF   bCounter =3 THEN 
				 			FOR j:=1 TO 4 BY 1 DO
									 FOR k:=1 TO 12 BY 1 DO
											 MEMCPY(ADR(arCameraResultHmi[5,j,k]),ADR(arCameraResultHmi[3,j,k]),SIZEOF(arCameraResultHmi[3,j,k]));
								END_FOR
							END_FOR	
					 END_IF	
					IF  bCounter =2 OR bCounter =3  THEN 
							FOR j:=1 TO 4 BY 1 DO
									 FOR k:=1 TO 12 BY 1 DO
											 MEMCPY(ADR(arCameraResultHmi[3,j,k]),ADR(arCameraResultHmi[1,j,k]),SIZEOF(arCameraResultHmi[1,j,k]));
											 MEMCPY(ADR(arCameraResultHmi[4,j,k]),ADR(arCameraResultHmi[2,j,k]),SIZEOF(arCameraResultHmi[2,j,k]));
											 MEMSET(ADR(arCameraResultHmi[1,j,k]),0,SIZEOF(arCameraResultHmi[1,j,k]));	
											 MEMSET(ADR(arCameraResultHmi[2,j,k]),0,SIZEOF(arCameraResultHmi[2,j,k]));	
								END_FOR
							END_FOR	
					END_IF
			
			
					station.iStepAuto:= 50;			
		50:////Restore_after_Estop_Process2/3 X轴位置1/2拍照流程
			 IF  station.xSingleRunning OR fbMachine[1].xTryRun THEN
					 station.iStepAuto :=70; 
			 ELSIF tsModuleProcess[bXCounter+1].xProcessNotStarted AND NOT  tsModuleProcess[bXCounter+1].xProcessStarted THEN
					 station.iStepAuto :=70; (*process not started*)
			 ELSIF  tsModuleProcess[bXCounter+1].xProcessStarted AND NOT  tsModuleProcess[bXCounter+1].xProcessCompleted THEN
					station.iStepAuto := 70;(*process started*)
			 ELSIF  tsModuleProcess[bXCounter+1].xProcessCompleted AND NOT tsModuleProcess[bXCounter+1].xQDataCompleted  THEN
					 station.iStepAuto :=200;(*process completed*)
			 ELSIF tsModuleProcess[bXCounter+1].xQDataCompleted THEN
					 station.iStepAuto :=200;(*Qdata completed *)
			 ELSE
					 station.iStepAuto :=70; 
			 END_IF	
		70://流程未开始
				tsModuleProcess[bXCounter+1].xProcessNotStarted :=TRUE;
				station.iStepAuto :=80; 
		80://水平调整气缸伸出		
			IF   bCounter =1 THEN
					IF  iBoxChoose =1 THEN
						(*上层水平调整气缸*)
						fbHOZAdjustCyl_1.xAuto :=TRUE;
						fbHOZAdjustCyl_2.xAuto :=TRUE;
						IF  fbHOZAdjustCyl_1.xWP_Delay  AND fbHOZAdjustCyl_2.xWP_Delay  THEN
								station.iStepAuto:= 90;
						END_IF
					ELSIF  iBoxChoose= 2 THEN
						(*下层水平调整气缸*)
						fbHOZAdjustCyl_3.xAuto :=TRUE;
						fbHOZAdjustCyl_4.xAuto :=TRUE;
						IF  fbHOZAdjustCyl_3.xWP_Delay AND fbHOZAdjustCyl_4.xWP_Delay  THEN
								station.iStepAuto:= 90;
						END_IF
					END_IF
			ELSIF  bCounter =2 OR  bCounter =3 OR bEndCounter =1 OR bEndCounter =2 THEN
					IF  iBoxChoose =1 THEN
						(*上层水平调整气缸*)
						IF   bEndCounter =0 THEN
							 fbHOZAdjustCyl_1.xAuto :=TRUE;
							 fbHOZAdjustCyl_2.xAuto :=TRUE;
						END_IF
						fbHOZAdjustCyl_5.xAuto :=TRUE;
						fbHOZAdjustCyl_6.xAuto :=TRUE;
						IF ( (fbHOZAdjustCyl_1.xWP_Delay  AND 
								fbHOZAdjustCyl_2.xWP_Delay ) OR  bEndCounter >0) AND
								 fbHOZAdjustCyl_5.xWP_Delay AND
								 fbHOZAdjustCyl_6.xWP_Delay THEN
								station.iStepAuto:= 90;
						END_IF
					ELSIF  iBoxChoose= 2 THEN
						(*下层水平调整气缸*)
						IF   bEndCounter =0 THEN
							 fbHOZAdjustCyl_3.xAuto :=TRUE;
							 fbHOZAdjustCyl_4.xAuto :=TRUE;
						END_IF
						fbHOZAdjustCyl_7.xAuto :=TRUE;
						fbHOZAdjustCyl_8.xAuto :=TRUE;
						IF  ((fbHOZAdjustCyl_3.xWP_Delay AND 
								fbHOZAdjustCyl_4.xWP_Delay ) OR  bEndCounter >0) AND 
								fbHOZAdjustCyl_7.xWP_Delay AND 
								fbHOZAdjustCyl_8.xWP_Delay  THEN
								station.iStepAuto:= 90;
						END_IF
					END_IF
			END_IF
		90://Z轴下降
			fbZAxisMove.xMoveAuto[2]:=TRUE;
			IF  fbZAxisMove.xMoveInPos[2] THEN
				station.iStepAuto:= 95;
			END_IF			 
		95://X轴移动到拍照位置1/2,Y轴到拍照位置1
				fbXAxisMove.xMoveAuto[bXCounter+1]:=TRUE;
				fbYAxisMove.xMoveAuto[2]:=TRUE;
				IF  fbXAxisMove.xMoveInPos[bXCounter+1]  AND 
					  fbYAxisMove.xMoveInPos[2]   THEN
					station.iStepAuto:= 100;
				END_IF
			
		100://设定Y轴循环开始 总次数为3
				 bYCounter:=1;
				station.iStepAuto:= 110;	
		110://Y轴移动到位置1/2/3	
				fbYAxisMove.xMoveAuto[bYCounter+1]:=TRUE;
				IF  fbYAxisMove.xMoveInPos[bYCounter+1] THEN
					station.iStepAuto:= 120;
				END_IF
		120://屏蔽拍照
			IF axBypassSignal[3] OR  fbMachine[1].xTryRun THEN
 					station.iStepAuto:= 150;	
			ELSE
					station.iStepAuto:= 140;		
			END_IF
		140://触发拍照
			(*开始循环*)
			tsModuleProcess[bXCounter+1].xProcessStarted :=TRUE;
			IF   bCounter =1  (*17.18位置有产品*)  THEN
							IF  bXCounter =1 THEN
									FOR i:=2 TO  9 BY 1 DO
										fbCamera[i].xlTrigger:=TRUE;
									END_FOR
							ELSIF bXCounter =2 THEN
									FOR i:=2 TO  5 BY 1 DO
										fbCamera[i].xlTrigger:=TRUE;
									END_FOR
							END_IF
			ELSIF  bCounter=2  THEN
							IF  bXCounter =1 THEN
										FOR i:=2 TO 17 BY 1 DO
											fbCamera[i].xlTrigger:=TRUE;
										END_FOR
							ELSIF   bXCounter =2 THEN
										FOR i:=2 TO 13 BY 1 DO
											fbCamera[i].xlTrigger:=TRUE;
										END_FOR	
							END_IF
			ELSIF   bCounter=3 THEN
							FOR i:=2 TO 17 BY 1 DO
								fbCamera[i].xlTrigger:=TRUE;
							END_FOR
			(*结束循环*)
			ELSIF   bEndCounter =1 (*17.18位置无产品*)  THEN
							IF  bXCounter =1 THEN
										FOR i:=6 TO  17 BY 1 DO
											fbCamera[i].xlTrigger:=TRUE;
										END_FOR
							ELSIF bXCounter =2 THEN
										FOR i:=2 TO  17 BY 1 DO
											fbCamera[i].xlTrigger:=TRUE;
										END_FOR
							END_IF
			ELSIF  bEndCounter =2 THEN
							IF  bXCounter =2 THEN
									FOR i:=14 TO  17 BY 1 DO
											fbCamera[i].xlTrigger:=TRUE;
									END_FOR	
							END_IF
			END_IF
			arTonDelay[07](IN:=FALSE);
			station.iStepAuto:=145;
	145://等待相机触发
				arTonDelay[07](IN:=TRUE , PT:=T#100MS , Q=> , ET=> );
				IF	 arTonDelay[07].Q THEN
				 		arTonDelay[07](IN:=FALSE);
				 		station.iStepAuto:=150;
				END_IF
	150://检查相机完成信号并储存
		(*开始循环*)
{region "bCounter =1 and bXCounter =1"}
			 IF   bCounter =1 (*17.18位置有产品*)  THEN	
				  	IF  bXCounter =1 THEN
								IF   axBypassSignal[3] OR  fbMachine[1].xTryRun THEN
													arMainlineFixtureData[arCurFixtureNumStation[5]].stProcessData.arCameraResult[3,bYCounter]:=
													arCameraResultHmi[1,3,bYCounter]:=1;	
													arMainlineFixtureData[arCurFixtureNumStation[5]].stProcessData.arCameraResult[3,6+bYCounter]:=
													arCameraResultHmi[1,3,6+bYCounter]:=1;	
													arMainlineFixtureData[arCurFixtureNumStation[5]].stProcessData.arCameraResult[1,3+bYCounter]:=
													arCameraResultHmi[1,1,3+bYCounter]:=1;
													arMainlineFixtureData[arCurFixtureNumStation[5]].stProcessData.arCameraResult[1,9+bYCounter]:=
													arCameraResultHmi[1,1,9+bYCounter]:=1;
													arProcessDataStation[2].stProcessData.arCameraResult[4,bYCounter]:=
													arCameraResultHmi[2,4,bYCounter]:=1;
													arProcessDataStation[2].stProcessData.arCameraResult[4,6+bYCounter]:=
													arCameraResultHmi[2,4,6+bYCounter]:=1;
													arProcessDataStation[2].stProcessData.arCameraResult[2,3+bYCounter]:=
													arCameraResultHmi[2,2,3+bYCounter]:=1;
													 arProcessDataStation[2].stProcessData.arCameraResult[2,9+bYCounter]:=
													arCameraResultHmi[2,2,9+bYCounter]:=1;	
													station.iStepAuto:=160;
								ELSE
										CASE  bResultStep OF
												0: //
														i_i_Counter:=1;
														bResultStep:=bResultStep +1;
												1://等待相机完成
														IF  fbCamera[i_i_Counter+1].xQDone THEN
																IF  i_i_Counter =1 THEN
																	arMainlineFixtureData[arCurFixtureNumStation[5]].stProcessData.arCameraResult[3,bYCounter]:=																	
																arCameraResultHmi[1,3,bYCounter]:=sCamera_To_Plc.iS03Result[i_i_Counter];	
															 ELSIF i_i_Counter =2 THEN
																 arMainlineFixtureData[arCurFixtureNumStation[5]].stProcessData.arCameraResult[3,6+bYCounter]:=
																 arCameraResultHmi[1,3,6+bYCounter]:=sCamera_To_Plc.iS03Result[i_i_Counter];	
															 ELSIF i_i_Counter =3 THEN
																 arMainlineFixtureData[arCurFixtureNumStation[5]].stProcessData.arCameraResult[1,3+bYCounter]:=
																 arCameraResultHmi[1,1,3+bYCounter]:=sCamera_To_Plc.iS03Result[i_i_Counter];
															 ELSIF i_i_Counter =4 THEN
																 arMainlineFixtureData[arCurFixtureNumStation[5]].stProcessData.arCameraResult[1,9+bYCounter]:=
																 arCameraResultHmi[1,1,9+bYCounter]:=sCamera_To_Plc.iS03Result[i_i_Counter];
															 ELSIF i_i_Counter =5 THEN
																	arProcessDataStation[2].stProcessData.arCameraResult[4,bYCounter]:= 
																 arCameraResultHmi[2,4,bYCounter]:=sCamera_To_Plc.iS03Result[i_i_Counter];
															 ELSIF i_i_Counter =6 THEN
																 arProcessDataStation[2].stProcessData.arCameraResult[4,6+bYCounter]:=
																 arCameraResultHmi[2,4,6+bYCounter]:=sCamera_To_Plc.iS03Result[i_i_Counter];
															 ELSIF i_i_Counter =7 THEN
																 arProcessDataStation[2].stProcessData.arCameraResult[2,3+bYCounter]:=
																 arCameraResultHmi[2,2,3+bYCounter]:=sCamera_To_Plc.iS03Result[i_i_Counter];
															 ELSIF i_i_Counter =8 THEN
																 arProcessDataStation[2].stProcessData.arCameraResult[2,9+bYCounter]:=
																 arCameraResultHmi[2,2,9+bYCounter]:=sCamera_To_Plc.iS03Result[i_i_Counter];	
															 END_IF	
															 bResultStep:=bResultStep +1;
													ELSIF   fbCamera[i_i_Counter+1].xQAlarm THEN
																		bResultStep:=0;
																		fbCamera[i_i_Counter+1].xlInit:=TRUE;
																		station.iStepAuto:=140;
																		station.adwAlarm[1].18	:=	TRUE;//	S03液位检测工位-相机检测超时报警,请检查
													END_IF
												2://循环计数
														 IF  i_i_Counter <8 THEN
																	i_i_Counter:=i_i_Counter+1;
																	bResultStep:=1;
														 ELSE
																
																bResultStep:=0;
																station.iStepAuto:=160;
														 END_IF											
										 END_CASE
								END_IF
					
{endregion}
{region "bCounter =1 and bXCounter =2"}
				 	ELSIF   bXCounter =2 THEN
									IF   axBypassSignal[3] OR  fbMachine[1].xTryRun THEN
															 arProcessDataStation[2].stProcessData.arCameraResult[3,bYCounter]:=
															 arCameraResultHmi[2,3,bYCounter]:=1;	
															arProcessDataStation[2].stProcessData.arCameraResult[3,6+bYCounter]:=
															arCameraResultHmi[2,3,6+bYCounter]:=1;	
															arProcessDataStation[2].stProcessData.arCameraResult[1,3+bYCounter]:=
															arCameraResultHmi[2,1,3+bYCounter]:=1;
															arProcessDataStation[2].stProcessData.arCameraResult[1,9+bYCounter]:=
															arCameraResultHmi[2,1,9+bYCounter]:=1;
															station.iStepAuto:=160;
																	
									ELSE
														CASE  bResultStep OF
																 0: //
																		i_i_Counter:=1;
																		bResultStep:=bResultStep +1;
																1://等待相机完成
																		IF  fbCamera[i_i_Counter+1].xQDone THEN
																				 IF  i_i_Counter =1 THEN
																					 arProcessDataStation[2].stProcessData.arCameraResult[3,bYCounter]:=
																					 arCameraResultHmi[2,3,bYCounter]:=sCamera_To_Plc.iS03Result[i_i_Counter];	
																				 ELSIF	i_i_Counter =2 THEN
																					 arProcessDataStation[2].stProcessData.arCameraResult[3,6+bYCounter]:=
																					 arCameraResultHmi[2,3,6+bYCounter]:=sCamera_To_Plc.iS03Result[i_i_Counter];	
																				 ELSIF i_i_Counter =3 THEN
																					  arProcessDataStation[2].stProcessData.arCameraResult[1,3+bYCounter]:=
																					 arCameraResultHmi[2,1,3+bYCounter]:=sCamera_To_Plc.iS03Result[i_i_Counter];
																				 ELSIF i_i_Counter =4 THEN
																						arProcessDataStation[2].stProcessData.arCameraResult[1,9+bYCounter]:=
																					 	arCameraResultHmi[2,1,9+bYCounter]:=sCamera_To_Plc.iS03Result[i_i_Counter];
																				 END_IF
																			 bResultStep:=bResultStep +1;
																	ELSIF   fbCamera[i_i_Counter+1].xQAlarm THEN
																				bResultStep:=0;
																				fbCamera[i_i_Counter+1].xlInit:=TRUE;
																				station.iStepAuto:=140;
																				station.adwAlarm[1].18	:=	TRUE;//	S03液位检测工位-相机检测超时报警,请检查
																	END_IF
																2://循环计数
																		 IF  i_i_Counter <4 THEN
																					i_i_Counter:=i_i_Counter+1;
																					bResultStep:=1;
																		 ELSE
																			
																				bResultStep:=0;
																				station.iStepAuto:=160;
																		 END_IF											
														 END_CASE
									END_IF		
						END_IF
{endregion}
{region "bCounter =2 and bXCounter =1"}
			 ELSIF  bCounter=2 THEN
					IF bXCounter =1 THEN
										 IF   axBypassSignal[3] OR  fbMachine[1].xTryRun THEN
												 							arMainlineFixtureData[arCurFixtureNumStation[5]].stProcessData.arCameraResult[3,bYCounter]:=
																			arCameraResultHmi[1,3,bYCounter]:=1;
																			arMainlineFixtureData[arCurFixtureNumStation[5]].stProcessData.arCameraResult[3,6+bYCounter]:=
																			arCameraResultHmi[1,3,6+bYCounter]:=1;	
																			arMainlineFixtureData[arCurFixtureNumStation[5]].stProcessData.arCameraResult[1,3+bYCounter]:=
																			arCameraResultHmi[1,1,3+bYCounter]:=1;
																			arMainlineFixtureData[arCurFixtureNumStation[5]].stProcessData.arCameraResult[1,9+bYCounter]:=
																			arCameraResultHmi[1,1,9+bYCounter]:=1;
																			arMainlineFixtureData[arCurFixtureNumStation[6]].stProcessData.arCameraResult[4,bYCounter]:=
																			arCameraResultHmi[2,4,bYCounter]:=1;
																			arMainlineFixtureData[arCurFixtureNumStation[6]].stProcessData.arCameraResult[4,6+bYCounter]:=
																			arCameraResultHmi[2,4,6+bYCounter]:=1;
																			arMainlineFixtureData[arCurFixtureNumStation[6]].stProcessData.arCameraResult[2,3+bYCounter]:=
																			arCameraResultHmi[2,2,3+bYCounter]:=1;
																			arMainlineFixtureData[arCurFixtureNumStation[6]].stProcessData.arCameraResult[2,9+bYCounter]:=
																			arCameraResultHmi[2,2,9+bYCounter]:=1;	
																			arMainlineFixtureData[arCurFixtureNumStation[7]].stProcessData.arCameraResult[3,3+bYCounter]:=
																			arCameraResultHmi[3,3,3+bYCounter]:=1;	
																			arMainlineFixtureData[arCurFixtureNumStation[7]].stProcessData.arCameraResult[3,9+bYCounter]:=
																			arCameraResultHmi[3,3,9+bYCounter]:=1;	
																			arMainlineFixtureData[arCurFixtureNumStation[7]].stProcessData.arCameraResult[1,bYCounter]:=
																			arCameraResultHmi[3,1,bYCounter]:= 1;
																			arMainlineFixtureData[arCurFixtureNumStation[7]].stProcessData.arCameraResult[1,6+bYCounter]:=
																			arCameraResultHmi[3,1,6+bYCounter]:=1;
																			arMainlineFixtureData[arCurFixtureNumStation[8]].stProcessData.arCameraResult[4,3+bYCounter]:=
																			arCameraResultHmi[4,4,3+bYCounter]:=1;
																			arMainlineFixtureData[arCurFixtureNumStation[8]].stProcessData.arCameraResult[4,9+bYCounter]:=
																			arCameraResultHmi[4,4,9+bYCounter]:=1;
																			arMainlineFixtureData[arCurFixtureNumStation[8]].stProcessData.arCameraResult[2,bYCounter]:=
																			arCameraResultHmi[4,2,bYCounter]:=1;
																			arMainlineFixtureData[arCurFixtureNumStation[8]].stProcessData.arCameraResult[2,6+bYCounter]:=
																			arCameraResultHmi[4,2,6+bYCounter]:=1;	
																			station.iStepAuto:=160;
										 ELSE
																		 CASE  bResultStep OF
																						0: //
																							 i_i_Counter:=1;
																							 bResultStep:=bResultStep +1;
																					 1://等待相机完成
																							 IF  fbCamera[i_i_Counter+1].xQDone THEN
																										 IF  i_i_Counter =1 THEN
																											 arMainlineFixtureData[arCurFixtureNumStation[5]].stProcessData.arCameraResult[3,bYCounter]:=
																											 arCameraResultHmi[1,3,bYCounter]:=sCamera_To_Plc.iS03Result[i_i_Counter];	 
																										 ELSIF i_i_Counter =2 THEN 
																											 arMainlineFixtureData[arCurFixtureNumStation[5]].stProcessData.arCameraResult[3,6+bYCounter]:=
																											 arCameraResultHmi[1,3,6+bYCounter]:=sCamera_To_Plc.iS03Result[i_i_Counter];	 
																										 ELSIF i_i_Counter =3 THEN 
																											 arMainlineFixtureData[arCurFixtureNumStation[5]].stProcessData.arCameraResult[1,3+bYCounter]:=
																											 arCameraResultHmi[1,1,3+bYCounter]:=sCamera_To_Plc.iS03Result[i_i_Counter]; 
																										 ELSIF i_i_Counter =4 THEN 
																											 arMainlineFixtureData[arCurFixtureNumStation[5]].stProcessData.arCameraResult[1,9+bYCounter]:=
																											 arCameraResultHmi[1,1,9+bYCounter]:=sCamera_To_Plc.iS03Result[i_i_Counter]; 
																										 ELSIF i_i_Counter =5 THEN 
																											 arMainlineFixtureData[arCurFixtureNumStation[6]].stProcessData.arCameraResult[4,bYCounter]:=
																											 arCameraResultHmi[2,4,bYCounter]:=sCamera_To_Plc.iS03Result[i_i_Counter]; 
																										 ELSIF i_i_Counter =6 THEN
																											 arMainlineFixtureData[arCurFixtureNumStation[6]].stProcessData.arCameraResult[4,6+bYCounter]:=
																											 arCameraResultHmi[2,4,6+bYCounter]:=sCamera_To_Plc.iS03Result[i_i_Counter]; 
																										 ELSIF i_i_Counter =7 THEN 
																											 arMainlineFixtureData[arCurFixtureNumStation[6]].stProcessData.arCameraResult[2,3+bYCounter]:=
																											 arCameraResultHmi[2,2,3+bYCounter]:=sCamera_To_Plc.iS03Result[i_i_Counter]; 
																										 ELSIF i_i_Counter =8 THEN 
																											  arMainlineFixtureData[arCurFixtureNumStation[6]].stProcessData.arCameraResult[2,9+bYCounter]:=
																											 arCameraResultHmi[2,2,9+bYCounter]:=sCamera_To_Plc.iS03Result[i_i_Counter];	 
																										 ELSIF i_i_Counter =9 THEN 
																											 arMainlineFixtureData[arCurFixtureNumStation[7]].stProcessData.arCameraResult[3,3+bYCounter]:=
																											 arCameraResultHmi[3,3,3+bYCounter]:=sCamera_To_Plc.iS03Result[i_i_Counter];	 
																										 ELSIF i_i_Counter =10 THEN 
																											 arMainlineFixtureData[arCurFixtureNumStation[7]].stProcessData.arCameraResult[3,9+bYCounter]:=
																											 arCameraResultHmi[3,3,9+bYCounter]:=sCamera_To_Plc.iS03Result[i_i_Counter];	 
																										 ELSIF i_i_Counter =11 THEN	
																											 arMainlineFixtureData[arCurFixtureNumStation[7]].stProcessData.arCameraResult[1,bYCounter]:= 
																											 arCameraResultHmi[3,1,bYCounter]:=sCamera_To_Plc.iS03Result[i_i_Counter]; 
																										 ELSIF i_i_Counter =12 THEN 
																											 arMainlineFixtureData[arCurFixtureNumStation[7]].stProcessData.arCameraResult[1,6+bYCounter]:= 
																											 arCameraResultHmi[3,1,6+bYCounter]:=sCamera_To_Plc.iS03Result[i_i_Counter]; 
																										 ELSIF i_i_Counter =13 THEN 
																											 arMainlineFixtureData[arCurFixtureNumStation[8]].stProcessData.arCameraResult[4,3+bYCounter]:= 
																											 arCameraResultHmi[4,4,3+bYCounter]:=sCamera_To_Plc.iS03Result[i_i_Counter]; 
																										 ELSIF i_i_Counter =14 THEN 
																											 arMainlineFixtureData[arCurFixtureNumStation[8]].stProcessData.arCameraResult[4,9+bYCounter]:= 
																											 arCameraResultHmi[4,4,9+bYCounter]:=sCamera_To_Plc.iS03Result[i_i_Counter]; 
																										 ELSIF i_i_Counter =15 THEN 
																											 arMainlineFixtureData[arCurFixtureNumStation[8]].stProcessData.arCameraResult[2,bYCounter]:= 
																											 arCameraResultHmi[4,2,bYCounter]:=sCamera_To_Plc.iS03Result[i_i_Counter]; 
																										 ELSIF i_i_Counter =16 THEN 
																											arMainlineFixtureData[arCurFixtureNumStation[8]].stProcessData.arCameraResult[2,6+bYCounter]:= 
																											 arCameraResultHmi[4,2,6+bYCounter]:=sCamera_To_Plc.iS03Result[i_i_Counter];	 
																										 END_IF	 
																										bResultStep:=bResultStep +1;
																						 ELSIF   fbCamera[i_i_Counter+1].xQAlarm THEN
																									 bResultStep:=0;
																									 fbCamera[i_i_Counter+1].xlInit:=TRUE;
																									 station.iStepAuto:=140;
																									 station.adwAlarm[1].18	:=	TRUE;//	S03液位检测工位-相机检测超时报警,请检查
																						 END_IF
																					 2://循环计数
																								IF  i_i_Counter <16 THEN
																										 i_i_Counter:=i_i_Counter+1;
																										 bResultStep:=1;
																								ELSE
																									 bResultStep:=0;
																									 station.iStepAuto:=160;
																								END_IF											
																				END_CASE
										 END_IF
{endregion}		
{region "bCounter =2 and bXCounter =2"}
			   ELSIF bXCounter =2 THEN
							IF   axBypassSignal[3] OR  fbMachine[1].xTryRun THEN
											arMainlineFixtureData[arCurFixtureNumStation[6]].stProcessData.arCameraResult[3,bYCounter]:= 
											arCameraResultHmi[2,3,bYCounter]:=1;
											arMainlineFixtureData[arCurFixtureNumStation[6]].stProcessData.arCameraResult[3,6+bYCounter]:= 															           
											arCameraResultHmi[2,3,6+bYCounter]:=1;	  
											arMainlineFixtureData[arCurFixtureNumStation[6]].stProcessData.arCameraResult[1,3+bYCounter]:=   											
											arCameraResultHmi[2,1,3+bYCounter]:=1; 
    									arMainlineFixtureData[arCurFixtureNumStation[6]].stProcessData.arCameraResult[1,9+bYCounter]:=  		
											arCameraResultHmi[2,1,9+bYCounter]:=1;    
											arMainlineFixtureData[arCurFixtureNumStation[7]].stProcessData.arCameraResult[4,bYCounter]:=  	 											
											arCameraResultHmi[3,4,bYCounter]:=1;     
											arMainlineFixtureData[arCurFixtureNumStation[7]].stProcessData.arCameraResult[4,6+bYCounter]:=    											
											arCameraResultHmi[3,4,6+bYCounter]:=1;  
											arMainlineFixtureData[arCurFixtureNumStation[7]].stProcessData.arCameraResult[2,3+bYCounter]:=   											
											arCameraResultHmi[3,2,3+bYCounter]:=1;   
											arMainlineFixtureData[arCurFixtureNumStation[7]].stProcessData.arCameraResult[2,9+bYCounter]:=  											
											arCameraResultHmi[3,2,9+bYCounter]:=1;			
											arMainlineFixtureData[arCurFixtureNumStation[8]].stProcessData.arCameraResult[3,3+bYCounter]:=    											
											arCameraResultHmi[4,3,3+bYCounter]:=1;	 
											arMainlineFixtureData[arCurFixtureNumStation[8]].stProcessData.arCameraResult[3,9+bYCounter]:=   											
											arCameraResultHmi[4,3,9+bYCounter]:=1;	    	
											arMainlineFixtureData[arCurFixtureNumStation[8]].stProcessData.arCameraResult[1,bYCounter]:=  										
											arCameraResultHmi[4,1,bYCounter]:=1;  
											arMainlineFixtureData[arCurFixtureNumStation[8]].stProcessData.arCameraResult[1,6+bYCounter]:=  	     											
											arCameraResultHmi[4,1,6+bYCounter]:=1;     											
											station.iStepAuto:=160;
							ELSE
												 CASE  bResultStep OF
															0: //
																 i_i_Counter:=1;
																 bResultStep:=bResultStep +1;
														 1://等待相机完成
																 IF  fbCamera[i_i_Counter+1].xQDone THEN
																			 	 IF  i_i_Counter =1 THEN
																						arMainlineFixtureData[arCurFixtureNumStation[6]].stProcessData.arCameraResult[3,bYCounter]:= 
																						 arCameraResultHmi[2,3,bYCounter]:=sCamera_To_Plc.iS03Result[i_i_Counter];		
																					 ELSIF i_i_Counter =2 THEN   
																						arMainlineFixtureData[arCurFixtureNumStation[6]].stProcessData.arCameraResult[3,6+bYCounter]:=     		 
																						 arCameraResultHmi[2,3,6+bYCounter]:=sCamera_To_Plc.iS03Result[i_i_Counter];					
																					 ELSIF i_i_Counter =3 THEN  
																						 arMainlineFixtureData[arCurFixtureNumStation[6]].stProcessData.arCameraResult[1,3+bYCounter]:=      					 
																						 arCameraResultHmi[2,1,3+bYCounter]:=sCamera_To_Plc.iS03Result[i_i_Counter];							
																					 ELSIF i_i_Counter =4 THEN     
																						 arMainlineFixtureData[arCurFixtureNumStation[6]].stProcessData.arCameraResult[1,9+bYCounter]:=   								 
																						 arCameraResultHmi[2,1,9+bYCounter]:=sCamera_To_Plc.iS03Result[i_i_Counter];										
																					 ELSIF i_i_Counter =5 THEN  
																						 	arMainlineFixtureData[arCurFixtureNumStation[7]].stProcessData.arCameraResult[4,bYCounter]:=  	     											 
																						 arCameraResultHmi[3,4,bYCounter]:=sCamera_To_Plc.iS03Result[i_i_Counter];													
																					 ELSIF i_i_Counter =6 THEN 
																						 arMainlineFixtureData[arCurFixtureNumStation[7]].stProcessData.arCameraResult[4,6+bYCounter]:=    														 
																						 arCameraResultHmi[3,4,6+bYCounter]:=sCamera_To_Plc.iS03Result[i_i_Counter];																
																					 ELSIF i_i_Counter =7 THEN 
																						 arMainlineFixtureData[arCurFixtureNumStation[7]].stProcessData.arCameraResult[2,3+bYCounter]:=     																	 
																						 arCameraResultHmi[3,2,3+bYCounter]:=sCamera_To_Plc.iS03Result[i_i_Counter];																			
																					 ELSIF i_i_Counter =8 THEN      	
																						 arMainlineFixtureData[arCurFixtureNumStation[7]].stProcessData.arCameraResult[2,9+bYCounter]:= 																			 
																						 arCameraResultHmi[3,2,9+bYCounter]:=sCamera_To_Plc.iS03Result[i_i_Counter];																							
																					 ELSIF i_i_Counter =9 THEN 
																							arMainlineFixtureData[arCurFixtureNumStation[8]].stProcessData.arCameraResult[3,3+bYCounter]:=      																							 
																						 arCameraResultHmi[4,3,3+bYCounter]:=sCamera_To_Plc.iS03Result[i_i_Counter];																										
																					 ELSIF i_i_Counter =10 THEN     
																						 arMainlineFixtureData[arCurFixtureNumStation[8]].stProcessData.arCameraResult[3,9+bYCounter]:=  																										 
																						 arCameraResultHmi[4,3,9+bYCounter]:=sCamera_To_Plc.iS03Result[i_i_Counter];																													
																					 ELSIF i_i_Counter =11 THEN      	
																						 arMainlineFixtureData[arCurFixtureNumStation[8]].stProcessData.arCameraResult[1,bYCounter]:=																												 
																						 arCameraResultHmi[4,1,bYCounter]:=sCamera_To_Plc.iS03Result[i_i_Counter];																															
																					 ELSIF i_i_Counter =12 THEN      		
																						 arMainlineFixtureData[arCurFixtureNumStation[8]].stProcessData.arCameraResult[1,6+bYCounter]:= 																														 
																						 arCameraResultHmi[4,1,6+bYCounter]:=sCamera_To_Plc.iS03Result[i_i_Counter];																																		
																					 END_IF																																				 																																									 
																			bResultStep:=bResultStep +1;
															 ELSIF   fbCamera[i_i_Counter+1].xQAlarm THEN
																		 bResultStep:=0;
																		 fbCamera[i_i_Counter+1].xlInit:=TRUE;
																		 station.iStepAuto:=140;
																		 station.adwAlarm[1].18	:=	TRUE;//	S03液位检测工位-相机检测超时报警,请检查
															 END_IF
														 2://循环计数
																	IF  i_i_Counter <12 THEN
																			 i_i_Counter:=i_i_Counter+1;
																			 bResultStep:=1;
																	ELSE
																		 bResultStep:=0;
																		 station.iStepAuto:=160;
																	END_IF											
											END_CASE
							END_IF
				END_IF
{endregion}	
 {region	"bCounter =3 and bXCounter =1"}              
			ELSIF  bCounter =3 THEN
					IF bXCounter =1 THEN
							IF   axBypassSignal[3] OR  fbMachine[1].xTryRun THEN
											arMainlineFixtureData[arCurFixtureNumStation[5]].stProcessData.arCameraResult[3,bYCounter]:=
											arCameraResultHmi[1,3,bYCounter]:=	1;
											arMainlineFixtureData[arCurFixtureNumStation[5]].stProcessData.arCameraResult[3,6+bYCounter]:=	
											arCameraResultHmi[1,3,6+bYCounter]:=1;	
											arMainlineFixtureData[arCurFixtureNumStation[5]].stProcessData.arCameraResult[1,3+bYCounter]:=
											arCameraResultHmi[1,1,3+bYCounter]:=1;
											arMainlineFixtureData[arCurFixtureNumStation[5]].stProcessData.arCameraResult[1,9+bYCounter]:=
											arCameraResultHmi[1,1,9+bYCounter]:=1;
											arMainlineFixtureData[arCurFixtureNumStation[6]].stProcessData.arCameraResult[4,bYCounter]:=
											arCameraResultHmi[2,4,bYCounter]:=1;
											arMainlineFixtureData[arCurFixtureNumStation[6]].stProcessData.arCameraResult[4,6+bYCounter]:=
											arCameraResultHmi[2,4,6+bYCounter]:=1;
											arMainlineFixtureData[arCurFixtureNumStation[6]].stProcessData.arCameraResult[2,3+bYCounter]:=	 
											arCameraResultHmi[2,2,3+bYCounter]:=1;
											arMainlineFixtureData[arCurFixtureNumStation[6]].stProcessData.arCameraResult[2,9+bYCounter]:=
											arCameraResultHmi[2,2,9+bYCounter]:=1;	
											arMainlineFixtureData[arCurFixtureNumStation[7]].stProcessData.arCameraResult[3,3+bYCounter]:=	
											arCameraResultHmi[3,3,3+bYCounter]:=1;	
											arMainlineFixtureData[arCurFixtureNumStation[7]].stProcessData.arCameraResult[3,9+bYCounter]:=		
											arCameraResultHmi[3,3,9+bYCounter]:=1;	
											arMainlineFixtureData[arCurFixtureNumStation[7]].stProcessData.arCameraResult[1,bYCounter]:=	
											arCameraResultHmi[3,1,bYCounter]:=1;
											arMainlineFixtureData[arCurFixtureNumStation[7]].stProcessData.arCameraResult[1,6+bYCounter]:=
											arCameraResultHmi[3,1,6+bYCounter]:=1;
											arMainlineFixtureData[arCurFixtureNumStation[8]].stProcessData.arCameraResult[4,3+bYCounter]:=
											arCameraResultHmi[4,4,3+bYCounter]:=1;
											arMainlineFixtureData[arCurFixtureNumStation[8]].stProcessData.arCameraResult[4,9+bYCounter]:=
											arCameraResultHmi[4,4,9+bYCounter]:=1;
											arMainlineFixtureData[arCurFixtureNumStation[8]].stProcessData.arCameraResult[2,bYCounter]:=
											arCameraResultHmi[4,2,bYCounter]:=1;
											arMainlineFixtureData[arCurFixtureNumStation[8]].stProcessData.arCameraResult[2,6+bYCounter]:=
											arCameraResultHmi[4,2,6+bYCounter]:=1;	
											station.iStepAuto:=160;
							ELSE
							 		CASE  bResultStep OF
															0: //
																 i_i_Counter:=1;
																 bResultStep:=bResultStep +1;
														 1://等待相机完成
																 IF  fbCamera[i_i_Counter+1].xQDone THEN
																		IF  i_i_Counter =1 THEN
																				arMainlineFixtureData[arCurFixtureNumStation[5]].stProcessData.arCameraResult[3,bYCounter]:=
																			arCameraResultHmi[1,3,bYCounter]:=sCamera_To_Plc.iS03Result[i_i_Counter];	
																		ELSIF i_i_Counter =2 THEN  
																			arMainlineFixtureData[arCurFixtureNumStation[5]].stProcessData.arCameraResult[3,6+bYCounter]:=	
																			arCameraResultHmi[1,3,6+bYCounter]:=sCamera_To_Plc.iS03Result[i_i_Counter];	
																		ELSIF i_i_Counter =3 THEN   
																			arMainlineFixtureData[arCurFixtureNumStation[5]].stProcessData.arCameraResult[1,3+bYCounter]:= 
																			arCameraResultHmi[1,1,3+bYCounter]:=sCamera_To_Plc.iS03Result[i_i_Counter];
																		ELSIF i_i_Counter =4 THEN   
																			arMainlineFixtureData[arCurFixtureNumStation[5]].stProcessData.arCameraResult[1,9+bYCounter]:= 
																			arCameraResultHmi[1,1,9+bYCounter]:=sCamera_To_Plc.iS03Result[i_i_Counter];
																		ELSIF i_i_Counter =5 THEN   
																			arMainlineFixtureData[arCurFixtureNumStation[6]].stProcessData.arCameraResult[4,bYCounter]:= 
																			arCameraResultHmi[2,4,bYCounter]:=sCamera_To_Plc.iS03Result[i_i_Counter];
																		ELSIF i_i_Counter =6 THEN   
																			arMainlineFixtureData[arCurFixtureNumStation[6]].stProcessData.arCameraResult[4,6+bYCounter]:= 
																			arCameraResultHmi[2,4,6+bYCounter]:=sCamera_To_Plc.iS03Result[i_i_Counter];
																		ELSIF i_i_Counter =7 THEN 
																			arMainlineFixtureData[arCurFixtureNumStation[6]].stProcessData.arCameraResult[2,3+bYCounter]:=	     
																			arCameraResultHmi[2,2,3+bYCounter]:=sCamera_To_Plc.iS03Result[i_i_Counter];
																		ELSIF i_i_Counter =8 THEN  
																			arMainlineFixtureData[arCurFixtureNumStation[6]].stProcessData.arCameraResult[2,9+bYCounter]:=   
																			arCameraResultHmi[2,2,9+bYCounter]:=sCamera_To_Plc.iS03Result[i_i_Counter];	
																		ELSIF i_i_Counter =9 THEN  
																			arMainlineFixtureData[arCurFixtureNumStation[7]].stProcessData.arCameraResult[3,3+bYCounter]:=   
																			arCameraResultHmi[3,3,3+bYCounter]:=sCamera_To_Plc.iS03Result[i_i_Counter];	
																		ELSIF i_i_Counter =10 THEN   
																			arMainlineFixtureData[arCurFixtureNumStation[7]].stProcessData.arCameraResult[3,9+bYCounter]:=	 
																			arCameraResultHmi[3,3,9+bYCounter]:=sCamera_To_Plc.iS03Result[i_i_Counter];	
																		ELSIF i_i_Counter =11 THEN   
																			arMainlineFixtureData[arCurFixtureNumStation[7]].stProcessData.arCameraResult[1,bYCounter]:=	 
																			arCameraResultHmi[3,1,bYCounter]:=sCamera_To_Plc.iS03Result[i_i_Counter];
																		ELSIF i_i_Counter =12 THEN    
																			arMainlineFixtureData[arCurFixtureNumStation[7]].stProcessData.arCameraResult[1,6+bYCounter]:=
																			arCameraResultHmi[3,1,6+bYCounter]:=sCamera_To_Plc.iS03Result[i_i_Counter];
																		ELSIF i_i_Counter =13 THEN 
																			arMainlineFixtureData[arCurFixtureNumStation[8]].stProcessData.arCameraResult[4,3+bYCounter]:=   
																			arCameraResultHmi[4,4,3+bYCounter]:=sCamera_To_Plc.iS03Result[i_i_Counter];
																		ELSIF i_i_Counter =14 THEN   
																			arMainlineFixtureData[arCurFixtureNumStation[8]].stProcessData.arCameraResult[4,9+bYCounter]:= 
																			arCameraResultHmi[4,4,9+bYCounter]:=sCamera_To_Plc.iS03Result[i_i_Counter];
																		ELSIF i_i_Counter =15 THEN    
																			arMainlineFixtureData[arCurFixtureNumStation[8]].stProcessData.arCameraResult[2,bYCounter]:=
																			arCameraResultHmi[4,2,bYCounter]:=sCamera_To_Plc.iS03Result[i_i_Counter];
																		ELSIF i_i_Counter =16 THEN	
																			arMainlineFixtureData[arCurFixtureNumStation[8]].stProcessData.arCameraResult[2,6+bYCounter]:=   
																			arCameraResultHmi[4,2,6+bYCounter]:=sCamera_To_Plc.iS03Result[i_i_Counter];	
                                    END_IF																																								 
																			bResultStep:=bResultStep +1;
															 ELSIF   fbCamera[i_i_Counter+1].xQAlarm THEN
																		 bResultStep:=0;
																		 fbCamera[i_i_Counter+1].xlInit:=TRUE;
																		 station.iStepAuto:=140;
																		 station.adwAlarm[1].18	:=	TRUE;//	S03液位检测工位-相机检测超时报警,请检查
															 END_IF
														 2://循环计数
																	IF  i_i_Counter <16 THEN
																			 i_i_Counter:=i_i_Counter+1;
																			 bResultStep:=1;
																	ELSE
																		 bResultStep:=0;
																		 station.iStepAuto:=160;
																	END_IF											
											END_CASE
							END_IF
{endregion}
{region "bCounter =3 and bxCounter =2"}
					ELSIF bXCounter =2 THEN
							IF   axBypassSignal[3] OR  fbMachine[1].xTryRun THEN
											arMainlineFixtureData[arCurFixtureNumStation[6]].stProcessData.arCameraResult[3,bYCounter]:= 
											arCameraResultHmi[2,3,bYCounter]:=1;	
											arMainlineFixtureData[arCurFixtureNumStation[6]].stProcessData.arCameraResult[3,6+bYCounter]:=
											arCameraResultHmi[2,3,6+bYCounter]:=1;	
											arMainlineFixtureData[arCurFixtureNumStation[6]].stProcessData.arCameraResult[1,3+bYCounter]:=
											arCameraResultHmi[2,1,3+bYCounter]:=1;
											arMainlineFixtureData[arCurFixtureNumStation[6]].stProcessData.arCameraResult[1,9+bYCounter]:=
											arCameraResultHmi[2,1,9+bYCounter]:=1;
											arMainlineFixtureData[arCurFixtureNumStation[7]].stProcessData.arCameraResult[4,bYCounter]:=
											arCameraResultHmi[3,4,bYCounter]:=1;
											arMainlineFixtureData[arCurFixtureNumStation[7]].stProcessData.arCameraResult[4,6+bYCounter]:=
											arCameraResultHmi[3,4,6+bYCounter]:=1;
											arMainlineFixtureData[arCurFixtureNumStation[7]].stProcessData.arCameraResult[2,3+bYCounter]:=
											arCameraResultHmi[3,2,3+bYCounter]:=1;
											arMainlineFixtureData[arCurFixtureNumStation[7]].stProcessData.arCameraResult[2,9+bYCounter]:=
											arCameraResultHmi[3,2,9+bYCounter]:=1;
											arMainlineFixtureData[arCurFixtureNumStation[8]].stProcessData.arCameraResult[3,3+bYCounter]:=	
											arCameraResultHmi[4,3,3+bYCounter]:=1;	
											arMainlineFixtureData[arCurFixtureNumStation[8]].stProcessData.arCameraResult[3,9+bYCounter]:=	
											arCameraResultHmi[4,3,9+bYCounter]:=1;	
											arMainlineFixtureData[arCurFixtureNumStation[8]].stProcessData.arCameraResult[1,bYCounter]:=	
											arCameraResultHmi[4,1,bYCounter]:=1;
											arMainlineFixtureData[arCurFixtureNumStation[8]].stProcessData.arCameraResult[1,6+bYCounter]:=	
											arCameraResultHmi[4,1,6+bYCounter]:=1;
											arMainlineFixtureData[arCurFixtureNumStation[9]].stProcessData.arCameraResult[4,3+bYCounter]:=	
											arCameraResultHmi[5,4,3+bYCounter]:=1;
											arMainlineFixtureData[arCurFixtureNumStation[9]].stProcessData.arCameraResult[4,9+bYCounter]:=	
											arCameraResultHmi[5,4,9+bYCounter]:=1;
											arMainlineFixtureData[arCurFixtureNumStation[9]].stProcessData.arCameraResult[2,bYCounter]:=	
											arCameraResultHmi[5,2,bYCounter]:=1;
											arMainlineFixtureData[arCurFixtureNumStation[9]].stProcessData.arCameraResult[2,6+bYCounter]:=	
											arCameraResultHmi[5,2,6+bYCounter]:=1;	
											station.iStepAuto:=160;
							ELSE
							 				CASE  bResultStep OF
															0: //
																 i_i_Counter:=1;
																 bResultStep:=bResultStep +1;
														 1://等待相机完成
																 IF  fbCamera[i_i_Counter+1].xQDone THEN
																			IF  i_i_Counter=1 THEN
																				arMainlineFixtureData[arCurFixtureNumStation[6]].stProcessData.arCameraResult[3,bYCounter]:= 
                                    		arCameraResultHmi[2,3,bYCounter]:=sCamera_To_Plc.iS03Result[i_i_Counter];	
                                    	ELSIF i_i_Counter =2 THEN 
																				arMainlineFixtureData[arCurFixtureNumStation[6]].stProcessData.arCameraResult[3,6+bYCounter]:=  
                                    		arCameraResultHmi[2,3,6+bYCounter]:=sCamera_To_Plc.iS03Result[i_i_Counter];	
                                    	ELSIF i_i_Counter =3 THEN    
																				arMainlineFixtureData[arCurFixtureNumStation[6]].stProcessData.arCameraResult[1,3+bYCounter]:=
                                    		arCameraResultHmi[2,1,3+bYCounter]:=sCamera_To_Plc.iS03Result[i_i_Counter];
                                    	ELSIF i_i_Counter =4 THEN
																			  arMainlineFixtureData[arCurFixtureNumStation[6]].stProcessData.arCameraResult[1,9+bYCounter]:=     
                                    		arCameraResultHmi[2,1,9+bYCounter]:=sCamera_To_Plc.iS03Result[i_i_Counter];
                                    	ELSIF i_i_Counter =5 THEN   
																				arMainlineFixtureData[arCurFixtureNumStation[7]].stProcessData.arCameraResult[4,bYCounter]:=  
                                    		arCameraResultHmi[3,4,bYCounter]:=sCamera_To_Plc.iS03Result[i_i_Counter];
                                    	ELSIF i_i_Counter =6 THEN  
																				arMainlineFixtureData[arCurFixtureNumStation[7]].stProcessData.arCameraResult[4,6+bYCounter]:=  
                                    		arCameraResultHmi[3,4,6+bYCounter]:=sCamera_To_Plc.iS03Result[i_i_Counter];
                                    	ELSIF i_i_Counter =7 THEN
																				arMainlineFixtureData[arCurFixtureNumStation[7]].stProcessData.arCameraResult[2,3+bYCounter]:=   
                                    		arCameraResultHmi[3,2,3+bYCounter]:=sCamera_To_Plc.iS03Result[i_i_Counter];
                                    	ELSIF i_i_Counter =8 THEN  
																				arMainlineFixtureData[arCurFixtureNumStation[7]].stProcessData.arCameraResult[2,9+bYCounter]:=   
                                    		arCameraResultHmi[3,2,9+bYCounter]:=sCamera_To_Plc.iS03Result[i_i_Counter];	
                                    	ELSIF i_i_Counter =9 THEN  
																				arMainlineFixtureData[arCurFixtureNumStation[8]].stProcessData.arCameraResult[3,3+bYCounter]:=	  
                                    		arCameraResultHmi[4,3,3+bYCounter]:=sCamera_To_Plc.iS03Result[i_i_Counter];	
                                    	ELSIF i_i_Counter =10 THEN 
																				arMainlineFixtureData[arCurFixtureNumStation[8]].stProcessData.arCameraResult[3,9+bYCounter]:=	   
                                    		arCameraResultHmi[4,3,9+bYCounter]:=sCamera_To_Plc.iS03Result[i_i_Counter];	
                                    	ELSIF i_i_Counter =11 THEN 
																				arMainlineFixtureData[arCurFixtureNumStation[8]].stProcessData.arCameraResult[1,bYCounter]:=	   
                                    		arCameraResultHmi[4,1,bYCounter]:=sCamera_To_Plc.iS03Result[i_i_Counter];
                                    	ELSIF i_i_Counter =12 THEN
																				arMainlineFixtureData[arCurFixtureNumStation[8]].stProcessData.arCameraResult[1,6+bYCounter]:=	    
                                    		arCameraResultHmi[4,1,6+bYCounter]:=sCamera_To_Plc.iS03Result[i_i_Counter];
                                    	ELSIF i_i_Counter =13 THEN 
																				arMainlineFixtureData[arCurFixtureNumStation[9]].stProcessData.arCameraResult[4,3+bYCounter]:=	  
                                    		arCameraResultHmi[5,4,3+bYCounter]:=sCamera_To_Plc.iS03Result[i_i_Counter];
                                    	ELSIF i_i_Counter =14 THEN   
																				arMainlineFixtureData[arCurFixtureNumStation[9]].stProcessData.arCameraResult[4,9+bYCounter]:=	 
                                    		arCameraResultHmi[5,4,9+bYCounter]:=sCamera_To_Plc.iS03Result[i_i_Counter];
                                    	ELSIF i_i_Counter =15 THEN    
                                    		arMainlineFixtureData[arCurFixtureNumStation[9]].stProcessData.arCameraResult[2,bYCounter]:=	
                                    		arCameraResultHmi[5,2,bYCounter]:=sCamera_To_Plc.iS03Result[i_i_Counter];
                                    	ELSIF	i_i_Counter =16 THEN  
																				arMainlineFixtureData[arCurFixtureNumStation[9]].stProcessData.arCameraResult[2,6+bYCounter]:=	 
                                    		arCameraResultHmi[5,2,6+bYCounter]:=sCamera_To_Plc.iS03Result[i_i_Counter];	
                                    	END_IF	
																			bResultStep:=bResultStep +1;
															 ELSIF   fbCamera[i_i_Counter+1].xQAlarm THEN
																		 bResultStep:=0;
																		 fbCamera[i_i_Counter+1].xlInit:=TRUE;
																		 station.iStepAuto:=140;
																		 station.adwAlarm[1].18	:=	TRUE;//	S03液位检测工位-相机检测超时报警,请检查
															 END_IF
														 2://循环计数
																	IF  i_i_Counter <16 THEN
																			 i_i_Counter:=i_i_Counter+1;
																			 bResultStep:=1;
																	ELSE
																		 bResultStep:=0;
																		 station.iStepAuto:=160;
																	END_IF											
											END_CASE
						 END_IF		
					END_IF											 
{endregion}
{region "bEndCounter =1 and bXCounter =1"}
		(*结束循环*)
			ELSIF   bEndCounter =1 (*17.18位置无产品*)  THEN	
				  	IF  bXCounter =1 THEN
							IF   axBypassSignal[3] OR  fbMachine[1].xTryRun THEN
											arMainlineFixtureData[arCurFixtureNumStation[7]].stProcessData.arCameraResult[3,3+bYCounter]:=	
											arCameraResultHmi[3,3,3+bYCounter]:=1;
											arMainlineFixtureData[arCurFixtureNumStation[7]].stProcessData.arCameraResult[3,9+bYCounter]:=	
											arCameraResultHmi[3,3,9+bYCounter]:=1;
											arMainlineFixtureData[arCurFixtureNumStation[7]].stProcessData.arCameraResult[1,bYCounter]:=	
											arCameraResultHmi[3,1,bYCounter]:=1;
											arMainlineFixtureData[arCurFixtureNumStation[7]].stProcessData.arCameraResult[1,3+bYCounter]:=	
											arCameraResultHmi[3,1,3+bYCounter]:=1; 
											arMainlineFixtureData[arCurFixtureNumStation[8]].stProcessData.arCameraResult[4,3+bYCounter]:=                
											arCameraResultHmi[4,4,3+bYCounter]:=1;
											arMainlineFixtureData[arCurFixtureNumStation[8]].stProcessData.arCameraResult[4,9+bYCounter]:=    	
											arCameraResultHmi[4,4,9+bYCounter]:=1;
											arMainlineFixtureData[arCurFixtureNumStation[8]].stProcessData.arCameraResult[2,bYCounter]:=   
											arCameraResultHmi[4,2,bYCounter]:=1;
											arMainlineFixtureData[arCurFixtureNumStation[8]].stProcessData.arCameraResult[2,6+bYCounter]:=  
											arCameraResultHmi[4,2,6+bYCounter]:=1;
											station.iStepAuto:=160;
							ELSE
									CASE  bResultStep OF
															0: //
																 i_i_Counter:=9;
																 bResultStep:=bResultStep +1;
														 1://等待相机完成
																 IF  fbCamera[i_i_Counter+1].xQDone THEN
																				IF i_i_Counter =9 THEN
																					arMainlineFixtureData[arCurFixtureNumStation[7]].stProcessData.arCameraResult[3,3+bYCounter]:=	
																					arCameraResultHmi[3,3,3+bYCounter]:=sCamera_To_Plc.iS03Result[i_i_Counter];
																				ELSIF i_i_Counter =10 THEN  
																					arMainlineFixtureData[arCurFixtureNumStation[7]].stProcessData.arCameraResult[3,9+bYCounter]:=	 
																					arCameraResultHmi[3,3,9+bYCounter]:=sCamera_To_Plc.iS03Result[i_i_Counter];
																				ELSIF i_i_Counter =11 THEN  
																					arMainlineFixtureData[arCurFixtureNumStation[7]].stProcessData.arCameraResult[1,bYCounter]:=	 
																					arCameraResultHmi[3,1,bYCounter]:=sCamera_To_Plc.iS03Result[i_i_Counter];
																				ELSIF i_i_Counter =12 THEN
																					arMainlineFixtureData[arCurFixtureNumStation[7]].stProcessData.arCameraResult[1,3+bYCounter]:=	    
																					arCameraResultHmi[3,1,3+bYCounter]:=sCamera_To_Plc.iS03Result[i_i_Counter];
																				ELSIF i_i_Counter =13 THEN
																					arMainlineFixtureData[arCurFixtureNumStation[8]].stProcessData.arCameraResult[4,3+bYCounter]:=       
																					arCameraResultHmi[4,4,3+bYCounter]:=sCamera_To_Plc.iS03Result[i_i_Counter];
																				ELSIF i_i_Counter =14 THEN    
																					arMainlineFixtureData[arCurFixtureNumStation[8]].stProcessData.arCameraResult[4,9+bYCounter]:=   
																					arCameraResultHmi[4,4,9+bYCounter]:=sCamera_To_Plc.iS03Result[i_i_Counter];
																				ELSIF i_i_Counter =15 THEN    
																				  arMainlineFixtureData[arCurFixtureNumStation[8]].stProcessData.arCameraResult[2,bYCounter]:=  
																					arCameraResultHmi[4,2,bYCounter]:=sCamera_To_Plc.iS03Result[i_i_Counter];
																				ELSIF i_i_Counter =16 THEN  
																					arMainlineFixtureData[arCurFixtureNumStation[8]].stProcessData.arCameraResult[2,6+bYCounter]:=   
																					arCameraResultHmi[4,2,6+bYCounter]:=sCamera_To_Plc.iS03Result[i_i_Counter];
																				END_IF
																			bResultStep:=bResultStep +1;
															 ELSIF   fbCamera[i_i_Counter+1].xQAlarm THEN
																		 bResultStep:=0;
																		 fbCamera[i_i_Counter+1].xlInit:=TRUE;
																		 station.iStepAuto:=140;
																		 station.adwAlarm[1].18	:=	TRUE;//	S03液位检测工位-相机检测超时报警,请检查
															 END_IF
														 2://循环计数
																	IF  i_i_Counter <16 THEN
																			 i_i_Counter:=i_i_Counter+1;
																			 bResultStep:=1;
																	ELSE
																		 bResultStep:=0;
																		 station.iStepAuto:=160;
																	END_IF											
											END_CASE 
							END_IF
{endregion}
{region "bEndCounter =1 and bXCounter =2"}		
				 	ELSIF   bXCounter =2 THEN
							IF   axBypassSignal[3] OR  fbMachine[1].xTryRun THEN
											arMainlineFixtureData[arCurFixtureNumStation[7]].stProcessData.arCameraResult[4,bYCounter]:=  
											arCameraResultHmi[3,4,bYCounter]:=1;	
											arMainlineFixtureData[arCurFixtureNumStation[7]].stProcessData.arCameraResult[4,6+bYCounter]:=
											arCameraResultHmi[3,4,6+bYCounter]:=1;	
											arMainlineFixtureData[arCurFixtureNumStation[7]].stProcessData.arCameraResult[2,3+bYCounter]:=
											arCameraResultHmi[3,2,3+bYCounter]:=1;
											arMainlineFixtureData[arCurFixtureNumStation[7]].stProcessData.arCameraResult[2,9+bYCounter]:=
											arCameraResultHmi[3,2,9+bYCounter]:=1;
											arMainlineFixtureData[arCurFixtureNumStation[8]].stProcessData.arCameraResult[3,3+bYCounter]:=
											arCameraResultHmi[4,3,3+bYCounter]:=1;
											arMainlineFixtureData[arCurFixtureNumStation[8]].stProcessData.arCameraResult[3,9+bYCounter]:=	
											arCameraResultHmi[4,3,9+bYCounter]:=1;	
											arMainlineFixtureData[arCurFixtureNumStation[8]].stProcessData.arCameraResult[1,bYCounter]:=
											arCameraResultHmi[4,1,bYCounter]:=1;
											arMainlineFixtureData[arCurFixtureNumStation[8]].stProcessData.arCameraResult[1,6+bYCounter]:=
											arCameraResultHmi[4,1,6+bYCounter]:=1;		
											arMainlineFixtureData[arCurFixtureNumStation[9]].stProcessData.arCameraResult[4,3+bYCounter]:=
											arCameraResultHmi[5,4,3+bYCounter]:=1;	
											arMainlineFixtureData[arCurFixtureNumStation[9]].stProcessData.arCameraResult[4,9+bYCounter]:=
											arCameraResultHmi[5,4,9+bYCounter]:=1;	
											arMainlineFixtureData[arCurFixtureNumStation[9]].stProcessData.arCameraResult[2,bYCounter]:=
											arCameraResultHmi[5,2,bYCounter]:=1;
											arMainlineFixtureData[arCurFixtureNumStation[9]].stProcessData.arCameraResult[2,6+bYCounter]:=
											arCameraResultHmi[5,2,6+bYCounter]:=1;
											station.iStepAuto:=160;
							ELSE
											CASE  bResultStep OF
															0: //
																 i_i_Counter:=5;
																 bResultStep:=bResultStep +1;
														 1://等待相机完成
																 IF  fbCamera[i_i_Counter+1].xQDone THEN
																					 IF  i_i_Counter =5 THEN
																						 arMainlineFixtureData[arCurFixtureNumStation[7]].stProcessData.arCameraResult[4,bYCounter]:= 
																						 arCameraResultHmi[3,4,bYCounter]:=sCamera_To_Plc.iS03Result[i_i_Counter];	
																					 ELSIF i_i_Counter =6 THEN  
																					   arMainlineFixtureData[arCurFixtureNumStation[7]].stProcessData.arCameraResult[4,6+bYCounter]:=  
																						 arCameraResultHmi[3,4,6+bYCounter]:=sCamera_To_Plc.iS03Result[i_i_Counter];	
																					 ELSIF i_i_Counter =7 THEN  			
																						 arMainlineFixtureData[arCurFixtureNumStation[7]].stProcessData.arCameraResult[2,3+bYCounter]:=  
																						 arCameraResultHmi[3,2,3+bYCounter]:=sCamera_To_Plc.iS03Result[i_i_Counter];
																					 ELSIF i_i_Counter =8 THEN  
																						 arMainlineFixtureData[arCurFixtureNumStation[7]].stProcessData.arCameraResult[2,9+bYCounter]:=  
																						 arCameraResultHmi[3,2,9+bYCounter]:=sCamera_To_Plc.iS03Result[i_i_Counter];
																					 ELSIF  i_i_Counter =9 THEN 
																						 arMainlineFixtureData[arCurFixtureNumStation[8]].stProcessData.arCameraResult[3,3+bYCounter]:=   
																						 arCameraResultHmi[4,3,3+bYCounter]:=sCamera_To_Plc.iS03Result[i_i_Counter];	
																					 ELSIF i_i_Counter =10 THEN   
																						 arMainlineFixtureData[arCurFixtureNumStation[8]].stProcessData.arCameraResult[3,9+bYCounter]:=	 
																						 arCameraResultHmi[4,3,9+bYCounter]:=sCamera_To_Plc.iS03Result[i_i_Counter];	
																					 ELSIF i_i_Counter =11 THEN 
																						 arMainlineFixtureData[arCurFixtureNumStation[8]].stProcessData.arCameraResult[1,bYCounter]:=   
																						 arCameraResultHmi[4,1,bYCounter]:=sCamera_To_Plc.iS03Result[i_i_Counter];
																					 ELSIF i_i_Counter =12 THEN 
																						 arMainlineFixtureData[arCurFixtureNumStation[8]].stProcessData.arCameraResult[1,6+bYCounter]:= 
																						 arCameraResultHmi[4,1,6+bYCounter]:=sCamera_To_Plc.iS03Result[i_i_Counter];		
																					 ELSIF i_i_Counter=13 THEN 
																						 arMainlineFixtureData[arCurFixtureNumStation[9]].stProcessData.arCameraResult[4,3+bYCounter]:=
																						 arCameraResultHmi[5,4,3+bYCounter]:=sCamera_To_Plc.iS03Result[i_i_Counter];	
																					 ELSIF i_i_Counter =14 THEN
																						 arMainlineFixtureData[arCurFixtureNumStation[9]].stProcessData.arCameraResult[4,9+bYCounter]:=   
																						 arCameraResultHmi[5,4,9+bYCounter]:=sCamera_To_Plc.iS03Result[i_i_Counter];	
																					 ELSIF i_i_Counter =15 THEN
																						 arMainlineFixtureData[arCurFixtureNumStation[9]].stProcessData.arCameraResult[2,bYCounter]:=   
																						 arCameraResultHmi[5,2,bYCounter]:=sCamera_To_Plc.iS03Result[i_i_Counter];
																					 ELSIF i_i_Counter =16 THEN  
																						 arMainlineFixtureData[arCurFixtureNumStation[9]].stProcessData.arCameraResult[2,6+bYCounter]:=
																						 arCameraResultHmi[5,2,6+bYCounter]:=sCamera_To_Plc.iS03Result[i_i_Counter];
																					 END_IF																																																 
																			bResultStep:=bResultStep +1;
															 ELSIF   fbCamera[i_i_Counter+1].xQAlarm THEN
																		 bResultStep:=0;
																		 fbCamera[i_i_Counter+1].xlInit:=TRUE;
																		 station.iStepAuto:=140;
																		 station.adwAlarm[1].18	:=	TRUE;//	S03液位检测工位-相机检测超时报警,请检查
															 END_IF
														 2://循环计数
																	IF  i_i_Counter <16 THEN
																			 i_i_Counter:=i_i_Counter+1;
																			 bResultStep:=1;
																	ELSE
																		 bResultStep:=0;
																		 station.iStepAuto:=160;
																	END_IF											
											END_CASE 
							END_IF
					END_IF
{endregion}
{region "bEndCounter=2 and bXCounter =1"}
			ELSIF  bEndCounter=2 THEN
					IF  bXCounter =1 THEN
							station.iStepAuto:=160;//需要添加内容
{endregion}	
{region "bEndCounter=2 and bXCounter =1"}
					ELSIF bXCounter =2 THEN
							IF   axBypassSignal[3] OR  fbMachine[1].xTryRun THEN
												arMainlineFixtureData[arCurFixtureNumStation[9]].stProcessData.arCameraResult[4,3+bYCounter]:=
												arCameraResultHmi[5,4,3+bYCounter]:=1;	
											  arMainlineFixtureData[arCurFixtureNumStation[9]].stProcessData.arCameraResult[4,9+bYCounter]:=
												arCameraResultHmi[5,4,9+bYCounter]:=1;	
												arMainlineFixtureData[arCurFixtureNumStation[9]].stProcessData.arCameraResult[4,bYCounter]:=
												arCameraResultHmi[5,4,bYCounter]:=1;
												arMainlineFixtureData[arCurFixtureNumStation[9]].stProcessData.arCameraResult[4,6+bYCounter]:=
												arCameraResultHmi[5,4,6+bYCounter]:=1;
												station.iStepAuto:=160;
							ELSE
									CASE  bResultStep OF
															0: //
																 i_i_Counter:=13;
																 bResultStep:=bResultStep +1;
														 1://等待相机完成
																 IF  fbCamera[i_i_Counter+1].xQDone THEN
																					IF  i_i_Counter =13 THEN
																						
																					 arMainlineFixtureData[arCurFixtureNumStation[9]].stProcessData.arCameraResult[4,3+bYCounter]:=																				
																					 arCameraResultHmi[5,4,3+bYCounter]:=sCamera_To_Plc.iS03Result[i_i_Counter];	
																				 ELSIF i_i_Counter =14 THEN
																					 arMainlineFixtureData[arCurFixtureNumStation[9]].stProcessData.arCameraResult[4,9+bYCounter]:=
																					 arCameraResultHmi[5,4,9+bYCounter]:=sCamera_To_Plc.iS03Result[i_i_Counter];	
																				 ELSIF i_i_Counter =15 THEN
																					 arMainlineFixtureData[arCurFixtureNumStation[9]].stProcessData.arCameraResult[4,bYCounter]:=
																					 arCameraResultHmi[5,4,bYCounter]:=sCamera_To_Plc.iS03Result[i_i_Counter];
																				 ELSIF i_i_Counter =16 THEN
																					 arMainlineFixtureData[arCurFixtureNumStation[9]].stProcessData.arCameraResult[4,6+bYCounter]:=
																					 arCameraResultHmi[5,4,6+bYCounter]:=sCamera_To_Plc.iS03Result[i_i_Counter];
																				 END_IF																			 
																				bResultStep:=bResultStep +1;
															 ELSIF   fbCamera[i_i_Counter+1].xQAlarm THEN
																		 bResultStep:=0;
																		 fbCamera[i_i_Counter+1].xlInit:=TRUE;
																		 station.iStepAuto:=140;
																		 station.adwAlarm[1].18	:=	TRUE;//	S03液位检测工位-相机检测超时报警,请检查
															 END_IF
														 2://循环计数
																	IF  i_i_Counter <16 THEN
																			 i_i_Counter:=i_i_Counter+1;
																			 bResultStep:=1;
																	ELSE
																		 bResultStep:=0;
																		 station.iStepAuto:=160;
																	END_IF											
											END_CASE 
							END_IF								
						END_IF
			END_IF	
{endregion}	
		160://Y循环+1
			bYCounter :=bYCounter +1 ;
			station.iStepAuto:=180;
			
		180://判断循环次数是否已到
			IF   bYCounter<=3 THEN
				station.iStepAuto:=110;
			ELSE
				station.iStepAuto:=190; 
			END_IF
		190:///X轴拍照流程完成
				 tsModuleProcess[bXCounter+1].xProcessCompleted:=TRUE;
				 tsModuleProcess[bXCounter+1].xQDataCompleted:=TRUE;
					station.iStepAuto:=210; 
	//	200://Y轴回拍照位置1
	//			fbYAxisMove.xMoveAuto[2]:=TRUE;
	//			IF  fbYAxisMove.xMoveInPos[2] THEN
	//				station.iStepAuto:=210;
	//			END_IF
		210://X循环 +1 
			bXCounter :=bXCounter +1;
			station.iStepAuto:=220;
		220://X循环判断
			IF   bXCounter<=2 THEN
				station.iStepAuto:=50;
			ELSE
				station.iStepAuto:=230; 
			END_IF	
		230://Z轴上升
				fbZAxisMove.xMoveAuto[1]:=TRUE;
			IF  fbZAxisMove.xMoveInPos[1] THEN
					station.iStepAuto:= 240;
			END_IF
		240://水平调整气缸松开
					fbHOZAdjustCyl_1.xAuto:=FALSE;
					fbHOZAdjustCyl_2.xAuto:=FALSE;
					fbHOZAdjustCyl_3.xAuto:=FALSE;
					fbHOZAdjustCyl_4.xAuto:=FALSE;
					fbHOZAdjustCyl_5.xAuto:=false;
					fbHOZAdjustCyl_6.xAuto:=FALSE;
					fbHOZAdjustCyl_7.xAuto:=false;
					fbHOZAdjustCyl_8.xAuto:=FALSE;
			IF  fbHOZAdjustCyl_1.xHP_Delay AND 
					fbHOZAdjustCyl_2.xHP_Delay AND
					fbHOZAdjustCyl_3.xHP_Delay AND
					fbHOZAdjustCyl_4.xHP_Delay AND 
					fbHOZAdjustCyl_5.xHP_Delay AND 
					fbHOZAdjustCyl_6.xHP_Delay AND
					fbHOZAdjustCyl_7.xHP_Delay AND
					fbHOZAdjustCyl_8.xHP_Delay THEN
					station.iStepAuto:=260;	
				END_IF

		260:////Restore_after_Estop_Process4 数据传输流程
			IF  station.xSingleRunning  THEN //OR fbMachine[1].xTryRun THEN
						station.iStepAuto :=999;
			ELSIF tsModuleProcess[4].xProcessNotStarted AND NOT  tsModuleProcess[4].xProcessStarted THEN
					station.iStepAuto :=270; (*process not started*)
			ELSIF  tsModuleProcess[4].xProcessStarted AND NOT  tsModuleProcess[4].xProcessCompleted THEN
				 station.iStepAuto := 275;(*process started*)
			ELSIF  tsModuleProcess[4].xProcessCompleted AND NOT tsModuleProcess[4].xQDataCompleted  THEN
					station.iStepAuto :=350;(*process completed*)
			ELSIF tsModuleProcess[4].xQDataCompleted THEN
					station.iStepAuto :=360;(*Qdata completed *)
			ELSE
					station.iStepAuto :=270; 
			END_IF		
		270://		
				tsModuleProcess[4].xProcessNotStarted:=TRUE;
				station.iStepAuto :=280;
		280://汇总结果【4】
				FOR i:=1 TO 4 BY 1 DO
					FOR j :=1 TO 12 BY 1 DO 
						IF bCounter = 2 OR bCounter = 3 OR bEndCounter =1 THEN
							IF arMainlineFixtureData[arCurFixtureNumStation[8]].stProcessData.arCameraResult[i,j]<> 1 THEN
							 	arMainlineFixtureData[arCurFixtureNumStation[8]].xMaterialOnOff:=TRUE;//待删
								arMainlineFixtureData[arCurFixtureNumStation[8]].stProduct.xLidChecking_NOK:=TRUE;
								arMainlineFixtureData[arCurFixtureNumStation[8]].stProduct.xLidChecking_OK:=FALSE;
								EXIT;
							ELSIF   i=4 AND j =12 THEN
							 	arMainlineFixtureData[arCurFixtureNumStation[8]].xMaterialOnOff:=TRUE;//待删
								arMainlineFixtureData[arCurFixtureNumStation[8]].stProduct.xLidChecking_NOK:=FALSE;
								arMainlineFixtureData[arCurFixtureNumStation[8]].stProduct.xLidChecking_OK:=TRUE;
							END_IF
						END_IF
					END_FOR
				END_FOR
				station.iStepAuto:=290;
		290://汇总结果【5】	
				FOR i:=1 TO 4 BY 1 DO
					FOR j :=1 TO 12 BY 1 DO 
						IF bCounter = 3  OR bEndCounter =2 THEN
							IF arMainlineFixtureData[arCurFixtureNumStation[9]].stProcessData.arCameraResult[i,j]<>1 THEN
							 	 arMainlineFixtureData[arCurFixtureNumStation[9]].xMaterialOnOff:=TRUE;//待删
								 arMainlineFixtureData[arCurFixtureNumStation[9]].stProduct.xLidChecking_NOK:=TRUE;
							 	 arMainlineFixtureData[arCurFixtureNumStation[9]].stProduct.xLidChecking_OK:=FALSE;
								EXIT;
							ELSIF  i=4 AND j =12 THEN
							 	 arMainlineFixtureData[arCurFixtureNumStation[9]].xMaterialOnOff:=TRUE;//待删
								 arMainlineFixtureData[arCurFixtureNumStation[9]].stProduct.xLidChecking_NOK:=FALSE;
								 arMainlineFixtureData[arCurFixtureNumStation[9]].stProduct.xLidChecking_OK:=TRUE; 
							END_IF
						END_IF
					END_FOR
				END_FOR
				tsModuleProcess[4].xProcessCompleted:=TRUE;
				station.iStepAuto:=999;
	////产品流程结束
	999://----Single Run Finish----
		arManualNOKHmiButton[3]:=FALSE;
		station.iStepAuto :=1000;
		IF NOT station.xSingleContinuousRun THEN
			station.xSingleRunFlag:=FALSE;
		END_IF
		
